(* IEC 61131-3 sources: tuk_project/src/control_systems/implementation/Old, 7 files *)

(* ---- sorting_buffer_assembly.st ---- *)
(****************************************************************************************************************************)
(* SORTING FUNCTION BLOCK *)
(****************************************************************************************************************************)

FUNCTION_BLOCK sorting
  (*==========================================================================================*)
  (* INPUTS AND OUTPUTS *)
  (*==========================================================================================*)

  (* INPUT *)
  (*------------------------------------------------------------*)
  VAR_INPUT
    S_AL1 : BOOL;
    S_BIN_1 : BOOL;
    S_AL1_BL : BOOL;
    CS_AL1_W : INT;
    RUNNING : BOOL;
  END_VAR

  (* OUTPUT *)
  (*------------------------------------------------------------*)
  VAR_OUTPUT
    SB_AL1 : BOOL;
    PUWS_AL1_1_PLUS : BOOL;
    PUWS_AL1_1_RT : BOOL;
    CS_AL1_PLUS : BOOL;
  END_VAR

  (* PLACES *)
  (*------------------------------------------------------------*)
  VAR_EXTERNAL
    P0 : BOOL;
    P1 : BOOL;
    P2 : BOOL;
    P3 : BOOL;
    P4 : BOOL;
    PB : BOOL;
    P5 : BOOL;
    P6 : BOOL;
    BIN1 : BOOL;
    BIN2 : BOOL;
    P_LID : BOOL;
    P_BASE : BOOL;
    STABLE : BOOL;
  END_VAR

  (* OTHERS *)
  (*------------------------------------------------------------*)
  VAR
    timer_1_P2 : TON;
    timer_1_P3 : TON;
  END_VAR

  timer_1_P2(IN:= P2, PT:= T#1000ms);
  timer_1_P3(IN:= P3, PT:= T#1000ms);

  STABLE:= 0;

  IF NOT RUNNING THEN
    P0:= 1;
    P1:= 1;
    P2:= 0;
    P3:= 0;
    P4:= 0;
    PB:= 0;
    BIN1:= 1;
    BIN2:= 0;
    P5:= 0;
    P6:= 0;
    P_LID:= 0;
    P_BASE:= 0;
  END_IF;

  P0:= 1;

  (*==========================================================================================*)
  (* TRANSITIONS *)
  (*==========================================================================================*)
  WHILE STABLE= 0 DO
    STABLE:= 1;
    (*T0112*)
    IF P0 AND P1 AND S_AL1 AND NOT P2 THEN
      P0:= 0;
      P1:= 0;
      P2:= 1;
      STABLE:= 0;
    END_IF;

    (*T23*)
    IF P2 AND timer_1_P2.Q AND NOT P3 THEN
      P2:= 0;
      P3:= 1;
      STABLE:= 0;
    END_IF;

    (*T34*)
    IF P3 AND timer_1_P3.Q AND NOT P4 THEN
      P3:= 0;
      P4:= 1;
    END_IF;

    (*T4B*)
    IF P4 AND ( (CS_AL1_W < 200) OR (CS_AL1_W > 400) ) AND NOT PB THEN
      P4:= 0;
      PB:= 1;
      STABLE:= 0;
    END_IF;

    (*T4B2*)
    IF PB AND BIN1 AND S_BIN_1 AND NOT BIN2 AND NOT P1 THEN
      PB:= 0;
      BIN1:= 0;
      BIN2:= 1;
      P1:= 1;
      STABLE:= 0;
    END_IF;

    (*TB21*)
    IF BIN2 AND NOT S_BIN_1 AND NOT BIN1 THEN
      BIN2:= 0;
      BIN1:= 1;
      STABLE:= 0;
    END_IF;

    (*T45*)
    IF P4 AND ( (CS_AL1_W > 200) AND (CS_AL1_W <= 300) ) AND NOT P5 THEN
      P4:= 0;
      P5:= 1;
      STABLE:= 0;
    END_IF;

    (*T46*)
    IF P4 AND ( (CS_AL1_W > 300) AND (CS_AL1_W <= 400) ) AND NOT P6 THEN
      P4:= 0;
      P6:= 1;
      STABLE:= 0;
    END_IF;

    (*T57*)
    IF P5 AND S_AL1_BL AND NOT P_LID AND NOT P1 THEN
      P5:= 0;
      P_LID:= 1;
      P1:= 1;
      STABLE:= 0;
    END_IF;

    (*T67*)
    IF P6 AND S_AL1_BL AND NOT P_BASE AND NOT P1 THEN
      P6:= 0;
      P_BASE:= 1;
      P1:= 1;
      STABLE:= 0;
    END_IF;

  END_WHILE;

  (*==========================================================================================*)
  (* OUTPUTS *)
  (*==========================================================================================*)
  (*SET SB_AL1*)
  IF P3 OR P4 OR PB OR P5 OR P6 THEN
    SB_AL1:= 1;
  END_IF;
  (*RESET SB_AL1*)
  IF P1 OR P2 THEN
    SB_AL1:= 0;
  END_IF;

  (*SET PUWS_AL1_1_PLUS*)
  IF PB OR P5 OR P6 THEN
    PUWS_AL1_1_PLUS:= 1;
  END_IF;

  (*RESET PUWS_AL1_1_PLUS*)
  IF P1 OR P2 OR P3 OR P4 THEN
    PUWS_AL1_1_PLUS:= 0;
  END_IF;

  (*SET PUWS_AL1_1_RT*)
  IF P5 OR P6 THEN
    PUWS_AL1_1_RT:= 1;
  END_IF;

  (*RESET PUWS_AL1_1_RT*)
  IF P1 OR P2 OR P3 OR P4 OR PB THEN
    PUWS_AL1_1_RT:= 0;
  END_IF;

  (*SET CS_AL1_PLUS*)
  IF P1 OR P2 OR P5 OR P6 OR PB THEN
    CS_AL1_PLUS:= 1;
  END_IF;

  (*RESET CS_AL1_PLUS*)
  IF P3 OR P4 THEN
    CS_AL1_PLUS:= 0;
  END_IF;

END_FUNCTION_BLOCK

(****************************************************************************************************************************)
(* BASE BUFFER FUNCTION BLOCK *)
(****************************************************************************************************************************)

FUNCTION_BLOCK base_buffer
  (*==========================================================================================*)
  (* INPUTS AND OUTPUTS *)
  (*==========================================================================================*)

  (* INPUT *)
  (*------------------------------------------------------------*)
  VAR_INPUT
    S_AL1_B : BOOL;
    P_AL1_B_FT : BOOL;
    P_AL1_B_BK : BOOL;
    S_AL1_B1 : BOOL;
    S_AL1_B2 : BOOL;
    S_AL1_B3 : BOOL;
    S_AL1_LP : BOOL;
    RUNNING : BOOL;
  END_VAR

  (* OUTPUT *)
  (*------------------------------------------------------------*)
  VAR_OUTPUT
    P_AL1_B : BOOL;
    SB_AL1_B1 : BOOL;
    SB_AL1_B2 : BOOL;
    SB_AL1_B3 : BOOL;
    STABLE : BOOL;
  END_VAR

  (* PLACES *)
  (*------------------------------------------------------------*)
  VAR_EXTERNAL
    P_BASE : BOOL;
    PB1 : BOOL;
    PUSH_B : BOOL;
    PB2 : BOOL;
    PB23 : BOOL;
    PB3 : BOOL;
    PB4 : BOOL;
    PB5 : BOOL;
    PB6 : BOOL;
    PB7 : BOOL;
    PB8 : BOOL;
    PBF1 : BOOL;
    PBF2 : BOOL;
    PBF3 : BOOL;
    PBF4 : BOOL;
  END_VAR

  (* OTHERS *)
  (*------------------------------------------------------------*)
  VAR
    timer_1_TB1 : TON;
  END_VAR

  timer_1_TB1(IN:= PB1, PT:= T#900ms);

  STABLE:= 0;

  IF NOT RUNNING THEN
    P_BASE:= 0;
    PB1:= 0;
    PUSH_B:= 1;
    PB2:= 0;
    PB23:= 0;
    PB3:= 0;
    PB4:= 0;
    PB5:= 0;
    PB6:= 0;
    PB7:= 0;
    PB8:= 0;
    PBF1:=1;
    PBF2:=1;
    PBF3:=1;
    PBF4:=1;

  END_IF;

  (*==========================================================================================*)
  (* TRANSITIONS *)
  (*==========================================================================================*)
  WHILE STABLE= 0 DO
    STABLE:= 1;

    (*TB0*)
    IF P_BASE AND S_AL1_B AND NOT PB1 THEN
      P_BASE:=0;
      PB1:=1;
      STABLE:=0;
    END_IF;

    (*TB1*)
    IF PB1 AND PUSH_B AND timer_1_TB1.Q AND NOT PB2 THEN
      PB1:=0;
      PUSH_B:=0;
      PB2:=1;
      STABLE:=0;
    END_IF;

    (*TB23*)
    IF PB2 AND P_AL1_B_FT AND NOT PB23 THEN
      PB2:=0;
      PB23:=1;
      STABLE:=0;
    END_IF;

    (*TB2*)
    IF PB23 AND P_AL1_B_FT AND NOT PB3 THEN
      PB23:=0;
      PB3:=1;
      STABLE:=0;
    END_IF;

    (*TB3*)
    IF PB3 AND P_AL1_B_BK AND NOT PB4 AND NOT PUSH_B THEN
      PB3:=0;
      PB4:=1;
      PUSH_B:=1;
      STABLE:=0;
    END_IF;

    (*TB4*)
    IF PB4 AND PBF1 AND S_AL1_B1 AND NOT PB5 THEN
      PB4:=0;
      PBF1:=0;
      PB5:=1;
      STABLE:=0;
    END_IF;

    (*TB5*)
    IF PB5 AND PBF2 AND S_AL1_B2 AND NOT PB6 AND NOT PBF1 THEN
      PB5:=0;
      PBF2:=0;
      PB6:=1;
      PBF1:=1;
      STABLE:=0;
    END_IF;

    (*TB6*)
    IF PB6 AND PBF3 AND S_AL1_B3 AND  NOT PB7 AND NOT PBF2 THEN
      PB6:=0;
      PBF3:=0;
      PB7:=1;
      PBF2:=1;
      STABLE:=0;
    END_IF;

    (*TB7*)
    IF PB7 AND PBF4 AND S_AL1_LP AND NOT PB8 THEN
      PB7:=0;
      PBF4:=0;
      PB8:=1;
      STABLE:=0;
    END_IF;

  END_WHILE;

  (*==========================================================================================*)
  (* OUTPUTS *)
  (*==========================================================================================*)
  (*P_AL1_B*)
  IF PB2 OR PB23 THEN
    P_AL1_B:=1;
  END_IF;
  IF P_BASE OR PB1 OR PB3 THEN
    P_AL1_B:=0;
  END_IF;

  (*SB_AL1_B1*)
  IF PB5 THEN
    SB_AL1_B1:=1;
  END_IF;
  IF PBF1 THEN
    SB_AL1_B1:=0;
  END_IF;

  (*SB_AL1_B2*)
  IF PB6 THEN
    SB_AL1_B2:=1;
  END_IF;
  IF PBF2 THEN
    SB_AL1_B2:=0;
  END_IF;

  (*SB_AL1_B3*)
  IF PB7 THEN
    SB_AL1_B3:=1;
  END_IF;
  IF PBF3 THEN
    SB_AL1_B3:=0;
  END_IF;

END_FUNCTION_BLOCK

(****************************************************************************************************************************)
(* LID BUFFER FUNCTION BLOCK *)
(****************************************************************************************************************************)

FUNCTION_BLOCK lid_buffer
  (*==========================================================================================*)
  (* INPUTS AND OUTPUTS *)
  (*==========================================================================================*)

  (* INPUT *)
  (*------------------------------------------------------------*)
  VAR_INPUT
    S_AL1_L : BOOL;
    P_AL1_L_FT : BOOL;
    P_AL1_L_BK : BOOL;
    S_AL1_L1 : BOOL;
    S_AL1_L2 : BOOL;
    S_AL1_L3 : BOOL;
    S_AL1_RP : BOOL;
    RUNNING : BOOL;
  END_VAR

  (* OUTPUT *)
  (*------------------------------------------------------------*)
  VAR_OUTPUT
    P_AL1_L : BOOL;
    SB_AL1_L1 : BOOL;
    SB_AL1_L2 : BOOL;
    SB_AL1_L3 : BOOL;
    STABLE : BOOL;
  END_VAR

  (* PLACES *)
  (*------------------------------------------------------------*)
  VAR_EXTERNAL
    P_LID : BOOL;
    PL1 : BOOL;
    PUSH_L : BOOL;
    PL2 : BOOL;
    PL23 : BOOL;
    PL3 : BOOL;
    PL4 : BOOL;
    PL5 : BOOL;
    PL6 : BOOL;
    PL7 : BOOL;
    PL8 : BOOL;
    PLF1 : BOOL;
    PLF2 : BOOL;
    PLF3 : BOOL;
    PLF4 : BOOL;
  END_VAR

  (* OTHERS *)
  (*------------------------------------------------------------*)
  VAR
    timer_1_TL1 : TON;
  END_VAR

  timer_1_TL1(IN:= PL1, PT:= T#900ms);

  STABLE:= 0;

  IF NOT RUNNING THEN
    P_LID:= 0;
    PL1:= 0;
    PUSH_L:= 1;
    PL2:= 0;
    PL23:= 0;
    PL3:= 0;
    PL4:= 0;
    PL5:= 0;
    PL6:= 0;
    PL7:= 0;
    PL8:= 0;
    PLF1:=1;
    PLF2:=1;
    PLF3:=1;
    PLF4:=1;

  END_IF;

  (*==========================================================================================*)
  (* TRANSITIONS *)
  (*==========================================================================================*)
  WHILE STABLE= 0 DO
    STABLE:= 1;

    (*TL0*)
    IF P_LID AND S_AL1_L AND NOT PL1 THEN
      P_LID:=0;
      PL1:=1;
      STABLE:=0;
    END_IF;

    (*TL1*)
    IF PL1 AND PUSH_L AND timer_1_TL1.Q AND NOT PL2 THEN
      PL1:=0;
      PUSH_L:=0;
      PL2:=1;
      STABLE:=0;
    END_IF;

    (*TL23*)
    IF PL2 AND P_AL1_L_FT AND NOT PL23 THEN
      PL2:=0;
      PL23:=1;
      STABLE:=0;
    END_IF;

    (*TL2*)
    IF PL23 AND P_AL1_L_FT AND NOT PL3 THEN
      PL23:=0;
      PL3:=1;
      STABLE:=0;
    END_IF;

    (*TL3*)
    IF PL3 AND P_AL1_L_BK AND NOT PL4 AND NOT PUSH_L THEN
      PL3:=0;
      PL4:=1;
      PUSH_L:=1;
      STABLE:=0;
    END_IF;

    (*TL4*)
    IF PL4 AND PLF1 AND S_AL1_L1 AND NOT PL5 THEN
      PL4:=0;
      PLF1:=0;
      PL5:=1;
      STABLE:=0;
    END_IF;

    (*TL5*)
    IF PL5 AND PLF2 AND S_AL1_L2 AND NOT PL6 AND NOT PLF1 THEN
      PL5:=0;
      PLF2:=0;
      PL6:=1;
      PLF1:=1;
      STABLE:=0;
    END_IF;

    (*TL6*)
    IF PL6 AND PLF3 AND S_AL1_L3 AND  NOT PL7 AND NOT PLF2 THEN
      PL6:=0;
      PLF3:=0;
      PL7:=1;
      PLF2:=1;
      STABLE:=0;
    END_IF;

    (*TL7*)
    IF PL7 AND PLF4 AND S_AL1_RP AND NOT PL8 THEN
      PL7:=0;
      PLF4:=0;
      PL8:=1;
      STABLE:=0;
    END_IF;

  END_WHILE;

  (*==========================================================================================*)
  (* OUTPUTS *)
  (*==========================================================================================*)
  (*P_AL1_L*)
  IF PL2 OR PL23 THEN
    P_AL1_L:=1;
  END_IF;
  IF P_LID OR PL1 OR PL3 THEN
    P_AL1_L:=0;
  END_IF;

  (*SB_AL1_L1*)
  IF PL5 THEN
    SB_AL1_L1:=1;
  END_IF;
  IF PLF1 THEN
    SB_AL1_L1:=0;
  END_IF;

  (*SB_AL1_L2*)
  IF PL6 THEN
    SB_AL1_L2:=1;
  END_IF;
  IF PLF2 THEN
    SB_AL1_L2:=0;
  END_IF;

  (*SB_AL1_L3*)
  IF PL7 THEN
    SB_AL1_L3:=1;
  END_IF;
  IF PLF3 THEN
    SB_AL1_L3:=0;
  END_IF;

END_FUNCTION_BLOCK

(****************************************************************************************************************************)
(* ASSEMBLY FUNCTION BLOCK *)
(****************************************************************************************************************************)
FUNCTION_BLOCK assembly
  (*==========================================================================================*)
  (* INPUTS AND OUTPUTS *)
  (*==========================================================================================*)

  (* INPUT *)
  (*------------------------------------------------------------*)
  VAR_INPUT
    AL1_DETECTED : BOOL;
    AL1_X_POS : WORD;
    AL1_Y_POS : WORD;
    AL1_Z_POS : WORD;
    LP_AL1_CLAMPED : BOOL;
    LP_AL1_LIMIT : BOOL;
    RP_AL1_CLAMPED : BOOL;
    RUNNING : BOOL;
  END_VAR

  (* OUTPUT *)
  (*------------------------------------------------------------*)
  VAR_OUTPUT
    AL1_X_SET : WORD;
    AL1_Y_SET : WORD;
    AL1_Z_SET : WORD;
    AL1_GRAB : BOOL;
    RP_AL1_CLAMP : BOOL;
    LP_AL1_RAISE : BOOL;
    LP_AL1_CLAMP : BOOL;
    SB_AL1_B3 : BOOL;
    SB_AL1_L3 : BOOL;
    STABLE : BOOL;
  END_VAR

  (* PLACES *)
  (*------------------------------------------------------------*)
  VAR_EXTERNAL
    PA0 : BOOL;
    PA1 : BOOL;
    PA2 : BOOL;
    PA3 : BOOL;
    PA4 : BOOL;
    PA5 : BOOL;
    PA6 : BOOL;
    PA7 : BOOL;
    PA8 : BOOL;
    PA9 : BOOL;
    PA10 : BOOL;
    PA11 : BOOL;
    PA12 : BOOL;
    PA13 : BOOL;
    PB8 : BOOL;
    PB9 : BOOL;
    PL8 : BOOL;
    PL9 : BOOL;
    PBF3 : BOOL;
    PBF4 : BOOL;
    PLF3 : BOOL;
    PLF4 : BOOL;
  END_VAR

  (* OTHERS *)
  (*------------------------------------------------------------*)
  VAR
    timer_1 : TON;
  END_VAR

  timer_1(IN:= PL9, PT:= T#300ms);

  STABLE:= 0;

  IF NOT RUNNING THEN

    PB9:=0;
    PL9:=0;
    PA0:=1;
    PA1:=0;
    PA2:=0;
    PA3:=0;
    PA4:=0;
    PA5:=0;
    PA6:=0;
    PA7:=0;
    PA8:=0;
    PA9:=0;
    PA10:=0;
    PA11:=0;
    PA12:=0;
    PA13:=0;
  END_IF;

  (*==========================================================================================*)
  (* TRANSITIONS *)
  (*==========================================================================================*)
  WHILE STABLE=0 DO

    STABLE:=1;

    (*TB8*)
    IF PB8 AND LP_AL1_CLAMPED AND NOT PB9 THEN
      PB8:=0;
      PB9:=1;
      STABLE:=0;
    END_IF;

    (*TL8*)
    IF PL8 AND RP_AL1_CLAMPED AND NOT PL9 THEN
      PL8:=0;
      PL9:=1;
      STABLE:=0;
    END_IF;

    (*TA0*)
    IF PL9 AND timer_1.Q AND PA0 AND RP_AL1_CLAMPED AND NOT AL1_DETECTED AND NOT PA1 THEN
      PL9:=0;
      PA0:=0;
      PA1:=1;
      STABLE:=0;
    END_IF;

    (*TA1*)
    IF PA1 AND AL1_X_POS>798 AND AL1_X_POS<802 AND AL1_Y_POS>148 AND AL1_Y_POS<152 AND NOT PA2 THEN
      PA1:=0;
      PA2:=1;
      STABLE:=0;
    END_IF;

    (*TA2*)
    IF PA2 AND AL1_Z_POS>798 AND AL1_Z_POS<802 AND NOT PA3 THEN
      PA2:=0;
      PA3:=1;
      STABLE:=0;
    END_IF;

    (*TA3*)
    IF PA3 AND NOT RP_AL1_CLAMPED AND NOT PA4 THEN
      PA3:=0;
      PA4:=1;
      STABLE:=0;
    END_IF;

    (*TA4*)
    IF PA4 AND AL1_Z_POS>398 AND AL1_Z_POS<402 AND NOT PA5 AND NOT PLF3 AND NOT PLF4 THEN
      PA4:=0;
      PA5:=1;
      PLF3:=1;
      PLF4:=1;
      STABLE:=0;
    END_IF;

    (*TA5*)
    IF PA5 AND PB9 AND AL1_DETECTED AND LP_AL1_CLAMPED AND AL1_X_POS>208 AND AL1_X_POS<212 AND AL1_Y_POS>148 AND AL1_Y_POS<152 AND NOT PA6 THEN
      PA5:=0;
      PB9:=0;
      PA6:=1;
      STABLE:=0;
    END_IF;

    (*TA6*)
    IF PA6 AND AL1_Z_POS>810 AND AL1_Z_POS<820 AND NOT PA7 THEN
      PA6:=0;
      PA7:=1;
      STABLE:=0;
    END_IF;

    (*TA7*)
    IF PA7 AND AL1_Z_POS>398 AND AL1_Z_POS<402 AND NOT PA8 THEN
      PA7:=0;
      PA8:=1;
      STABLE:=0;
    END_IF;

    (*TA8*)
    IF PA8 AND NOT LP_AL1_CLAMPED AND NOT PA9 THEN
      PA8:=0;
      PA9:=1;
      STABLE:=0;
    END_IF;

    (*TA9*)
    IF PA9 AND NOT LP_AL1_LIMIT AND NOT PA10 THEN
      PA9:=0;
      PA10:=1;
      STABLE:=0;
    END_IF;

    (*TA10*)
    IF PA10 AND LP_AL1_LIMIT AND NOT PA11 THEN
      PA10:=0;
      PA11:=1;
      STABLE:=0;
    END_IF;

    (*TA11*)
    IF PA11 AND NOT LP_AL1_LIMIT AND NOT PA12 THEN
      PA11:=0;
      PA12:=1;
      STABLE:=0;
    END_IF;

    (*TA12*)
    IF PA12 AND LP_AL1_LIMIT AND NOT PA13 AND NOT PA0 AND NOT PBF3 AND NOT PBF4 THEN
      PA12:=0;
      PA13:=1;
      PA0:=1;
      PBF3:=1;
      PBF4:=1;
      STABLE:=0;
    END_IF;

  END_WHILE;

  (*==========================================================================================*)
  (* OUTPUTS *)
  (*==========================================================================================*)

  (*LP_AL1_CLAMP*)
  IF PB8 OR PB9 THEN
    LP_AL1_CLAMP:=1;
  END_IF;
  IF PBF4 THEN
    LP_AL1_CLAMP:=0;
  END_IF;

  (*RP_AL1_CLAMP*)
  IF PL8 OR PL9 THEN
    RP_AL1_CLAMP:=1;
  END_IF;
  IF PLF4 THEN
    RP_AL1_CLAMP:=0;
  END_IF;

  (*MOVE GRABBER TO LID POSITION*)
  IF PA1 THEN
    AL1_X_SET:=800;
    AL1_Y_SET:=150;
  END_IF;

  (*GRABBER DOWN TO PICK LID*)
  IF PA2 THEN
    AL1_Z_SET:= 800;
  END_IF;

  (*GRAB LID*)
  IF PA3 OR PA4 OR PA5 OR PA6 THEN
    AL1_GRAB:=1;
  END_IF;

  (*RAISE GRABBER A LITTLE*)
  IF PA0 OR PA4 OR PA7 THEN
    AL1_Z_SET:=400;
  END_IF;

  (*MOVE GRABBER TO BASE POSITION*)
  IF PA0 OR PA5 THEN
    AL1_X_SET:=210;
    AL1_Y_SET:=150;
  END_IF;

  (*LOWER LID TO FIT ON BASE*)
  IF PA6 THEN
    AL1_Z_SET:=818;
  END_IF;

  (*RELEASE LID*)
  IF PA0 OR PA1 OR PA2 OR PA7 OR PA8 OR PA9 OR PA10 OR PA11 OR PA12 THEN
    AL1_GRAB:=0;
  END_IF;

  (*LID CLAMP*)
  IF PA1 OR PA2 THEN
    RP_AL1_CLAMP:=1;
  END_IF;

  IF PA3 OR PA4 OR PLF4 THEN
    RP_AL1_CLAMP:=0;
  END_IF;

  (*BASE CLAMP*)
  IF PA8 OR PA9 OR PA10 OR PA11 OR PA12 THEN
    LP_AL1_CLAMP:=0;
  END_IF;

  IF PB9 OR PA6 OR PA7 THEN
    LP_AL1_CLAMP:=1;
  END_IF;

  (*RAISE BASE CLAMP*)
  IF PA0 OR PA1 OR PA2 OR PA3 OR PA4 OR PA5 OR PA6 OR PA7 OR PA8 OR PA11 OR PA12 THEN
    LP_AL1_RAISE:=0;
  END_IF;

  IF PA9 OR PA10 THEN
    LP_AL1_RAISE:=1;
  END_IF;

  (* OUTPUTS OF PLACES FROM OTHER STAGES *)
  (*LP_AL1_CLAMP*)
  (*IF PB9 THEN
    LP_AL1_CLAMP:=1;
  END_IF;
  IF PBF4 THEN
    LP_AL1_CLAMP:=0;
  END_IF;

  (*SB_AL1_B3
  IF PBF3 THEN
    SB_AL1_B3:=0;
  END_IF;

  (*SB_AL1_L3
  IF PLF3 THEN
    SB_AL1_L3:=0;
  END_IF;

  (*RP_AL1_CLAMP
  IF PL9 THEN
    RP_AL1_CLAMP:=1;
  END_IF;
  IF PLF4 THEN
    RP_AL1_CLAMP:=0;
  END_IF;  *)

END_FUNCTION_BLOCK

(****************************************************************************************************************************)
(* MAIN PROGRAM *)
(****************************************************************************************************************************)

PROGRAM sorting_buffer_assembly

  (****************************************************************************************************************************)
  (* VARIABLE DECLARATION *)
  (****************************************************************************************************************************)

  (*==========================================================================================*)
  (* INPUTS AND OUTPUTS *)
  (*==========================================================================================*)

  (* SORTING *)
  (*------------------------------------------------------------*)
  VAR
    (* INPUTS *)
    S_AL1 AT %IX102.0 : BOOL;
    S_BIN_1 AT %IX102.1 : BOOL;
    S_AL1_BL AT %IX102.2 : BOOL;
    CS_AL1_W AT %IW100 : INT;

    (* OUTPUTS *)
    SB_AL1 AT %QX101.2 : BOOL;
    PUWS_AL1_1_PLUS AT %QX101.3 : BOOL;
    PUWS_AL1_1_RT AT %QX101.4 : BOOL;
    CS_AL1_PLUS AT %QX101.5 : BOOL;
  END_VAR

  (* BUFFER *)
  (*------------------------------------------------------------*)
  VAR
    (* INPUTS *)
    S_AL1_B AT %IX100.0 : BOOL;
    P_AL1_B_FT AT %IX100.1 : BOOL;
    P_AL1_B_BK AT %IX100.2 : BOOL;
    S_AL1_B1 AT %IX100.3 : BOOL;
    S_AL1_B2 AT %IX100.4 : BOOL;
    S_AL1_B3 AT %IX100.5 : BOOL;
    LP_AL1_CLAMPED AT %IX100.6 : BOOL;
    S_AL1_LP AT %IX100.7 : BOOL;
    S_AL1_L AT %IX101.0 : BOOL;
    P_AL1_L_FT AT %IX101.1 : BOOL;
    P_AL1_L_BK AT %IX101.2 : BOOL;
    S_AL1_L1 AT %IX101.3 : BOOL;
    S_AL1_L2 AT %IX101.4 : BOOL;
    S_AL1_L3 AT %IX101.5 : BOOL;
    RP_AL1_CLAMPED AT %IX101.6 : BOOL;
    S_AL1_RP AT %IX101.7 : BOOL;

    (* OUTPUTS *)
    P_AL1_B AT %QX100.0 : BOOL;
    SB_AL1_B1 AT %QX100.1 : BOOL;
    SB_AL1_B2 AT %QX100.2 : BOOL;
    SB_AL1_B3 AT %QX100.3 : BOOL;
    LP_AL1_CLAMP AT %QX100.4 : BOOL;
    P_AL1_L AT %QX100.5 : BOOL;
    SB_AL1_L1 AT %QX100.6 : BOOL;
    SB_AL1_L2 AT %QX100.7 : BOOL;
    SB_AL1_L3 AT %QX101.0 : BOOL;
    RP_AL1_CLAMP AT %QX101.1 : BOOL;

  END_VAR

  (* ASSEMBLY *)
  (*------------------------------------------------------------*)
  VAR
    (* INPUTS *)
    AL1_DETECTED AT %IX102.3 : BOOL;
    LP_AL1_LIMIT AT %IX102.4 : BOOL;
    AL1_X_POS AT %IW101 : WORD;
    AL1_Y_POS AT %IW102 : WORD;
    AL1_Z_POS AT %IW103 : WORD;

    (* OUTPUTS *)
    AL1_GRAB AT %QX101.6 : BOOL;
    LP_AL1_RAISE AT %QX101.7 : BOOL;
    AL1_X_SET AT %QW100 : WORD;
    AL1_Y_SET AT %QW101 : WORD;
    AL1_Z_SET AT %QW102 : WORD;

  END_VAR

  (* OTHERS *)
  (*------------------------------------------------------------*)
  VAR
    (* RUNNING *)
    RUNNING AT %IX102.7 : BOOL;
  END_VAR

  (*==========================================================================================*)
  (* PLACES *)
  (*==========================================================================================*)
  (* ASSEMBLY *)
  (*------------------------------------------------------------*)
  VAR_EXTERNAL

    PA0 : BOOL;
    PA1 : BOOL;
    PA2 : BOOL;
    PA3 : BOOL;
    PA4 : BOOL;
    PA5 : BOOL;
    PA6 : BOOL;
    PA7 : BOOL;
    PA8 : BOOL;
    PA9 : BOOL;
    PA10 : BOOL;
    PA11 : BOOL;
    PA12 : BOOL;
    PA13 : BOOL;
    PL9 : BOOL;
    PB9 : BOOL;
    PBF3 : BOOL;
    PBF4 : BOOL;
    PLF3 : BOOL;
    PLF4 : BOOL;
  END_VAR
  (*==========================================================================================*)
  (* OTHERS *)
  (*==========================================================================================*)
  VAR_EXTERNAL
    STABLE : BOOL;
  END_VAR

  (****************************************************************************************************************************)
  (* VARIABLE INITIALIZATION *)
  (****************************************************************************************************************************)

  (*==========================================================================================*)
  (* FUNTION BLOCKS *)
  (*==========================================================================================*)
  VAR
    sorting0 : sorting;
    base_buffer0 : base_buffer;
    lid_buffer0 : lid_buffer;
    assembly0 : assembly;
  END_VAR

  (*==========================================================================================*)
  (* PLACES *)
  (*==========================================================================================*)

  (****************************************************************************************************************************)
  (* FUNCTION BLOCKS *)
  (****************************************************************************************************************************)

  (* SORTING *)
  (*------------------------------------------------------------*)
  sorting0(
    S_AL1:=S_AL1, S_BIN_1:=S_BIN_1, S_AL1_BL:=S_AL1_BL,
    CS_AL1_W:=CS_AL1_W, RUNNING:=RUNNING,

    SB_AL1=>SB_AL1, PUWS_AL1_1_PLUS=>PUWS_AL1_1_PLUS,
    PUWS_AL1_1_RT=>PUWS_AL1_1_RT, CS_AL1_PLUS=>CS_AL1_PLUS
  );

  (* BASE BUFFER *)
  (*------------------------------------------------------------*)
  base_buffer0(
    S_AL1_B:=S_AL1_B, P_AL1_B_FT:=P_AL1_B_FT, P_AL1_B_BK:=P_AL1_B_BK,
    S_AL1_B1:=S_AL1_B1, S_AL1_B2:=S_AL1_B2, S_AL1_B3:=S_AL1_B3,
    S_AL1_LP:=S_AL1_LP, (*LP_AL1_CLAMPED:=LP_AL1_CLAMPED,*) RUNNING:=RUNNING,

    P_AL1_B=>P_AL1_B, SB_AL1_B1=>SB_AL1_B1, SB_AL1_B2=>SB_AL1_B2,
    SB_AL1_B3=>SB_AL1_B3, STABLE=>STABLE (*, LP_AL1_CLAMP=>LP_AL1_CLAMP*)
  );

  (* LID BUFFER *)
  (*------------------------------------------------------------*)
  lid_buffer0(
    S_AL1_L:=S_AL1_L, P_AL1_L_FT:=P_AL1_L_FT, P_AL1_L_BK:=P_AL1_L_BK,
    S_AL1_L1:=S_AL1_L1, S_AL1_L2:=S_AL1_L2, S_AL1_L3:=S_AL1_L3,
    S_AL1_RP:=S_AL1_RP, (*RP_AL1_CLAMPED:=RP_AL1_CLAMPED,*) RUNNING:=RUNNING,

    P_AL1_L=>P_AL1_L, SB_AL1_L1=>SB_AL1_L1, SB_AL1_L2=>SB_AL1_L2,
    SB_AL1_L3=>SB_AL1_L3, STABLE=>STABLE (*, RP_AL1_CLAMP=>RP_AL1_CLAMP*)
  );

  (* ASSEMBLY *)
  (*------------------------------------------------------------*)
  assembly0(
    RP_AL1_CLAMPED:=RP_AL1_CLAMPED, AL1_DETECTED:=AL1_DETECTED,
    AL1_X_POS:=AL1_X_POS, AL1_Y_POS:=AL1_Y_POS, AL1_Z_POS:=AL1_Z_POS,
    LP_AL1_CLAMPED:=LP_AL1_CLAMPED, LP_AL1_LIMIT:=LP_AL1_LIMIT,
    RUNNING:=RUNNING,

    AL1_X_SET=>AL1_X_SET, AL1_Y_SET=>AL1_Y_SET, AL1_Z_SET=>AL1_Z_SET,
    AL1_GRAB=>AL1_GRAB, RP_AL1_CLAMP=>RP_AL1_CLAMP, LP_AL1_CLAMP=>LP_AL1_CLAMP,
    LP_AL1_RAISE=>LP_AL1_RAISE, STABLE=>STABLE (*,SB_AL1_B3=>SB_AL1_B3, SB_AL1_L3=>SB_AL1_L3*)
  );

END_PROGRAM

CONFIGURATION Config0

  (*==========================================================================================*)
  (* PLACES *)
  (*==========================================================================================*)

  (* SORTING *)
  (*------------------------------------------------------------*)
  VAR_GLOBAL
    P0 AT %QX103.0 : BOOL;
    P1 AT %QX103.1 : BOOL;
    P2 AT %QX103.2 : BOOL;
    P3 AT %QX103.3 : BOOL;
    P4 AT %QX103.4 : BOOL;
    PB AT %QX103.5 : BOOL;
    P5 AT %QX103.6 : BOOL;
    P6 AT %QX103.7 : BOOL;
    BIN1 AT %QX104.0 : BOOL;
    BIN2 AT %QX104.1 : BOOL;
    P_LID AT %QX104.2 : BOOL;
    P_BASE AT %QX104.3 : BOOL;
  END_VAR

  (* BUFFER *)
  (*------------------------------------------------------------*)
  VAR_GLOBAL
    PB1 AT %QX105.1 : BOOL;
    PUSH_B AT %QX105.2 : BOOL;
    PB2 AT %QX105.3 : BOOL;
    PB23 AT %QX105.4 : BOOL;
    PB3 AT %QX105.5 : BOOL;
    PB4 AT %QX105.6 : BOOL;
    PB5 AT %QX105.7 : BOOL;
    PB6 AT %QX106.0 : BOOL;
    PB7 AT %QX106.1 : BOOL;
    PB8 AT %QX106.2 : BOOL;
    PB9 AT %QX106.3 : BOOL;
    PBF1 AT %QX106.4 : BOOL;
    PBF2 AT %QX106.5 : BOOL;
    PBF3 AT %QX106.6 : BOOL;
    PBF4 AT %QX106.7 : BOOL;
    PL1 AT %QX107.1 : BOOL;
    PL2 AT %QX107.2 : BOOL;
    PUSH_L AT %QX107.3 : BOOL;
    PL23 AT %QX107.4 : BOOL;
    PL3 AT %QX107.5 : BOOL;
    PL4 AT %QX107.6 : BOOL;
    PL5 AT %QX107.7 : BOOL;
    PL6 AT %QX108.0 : BOOL;
    PL7 AT %QX108.1 : BOOL;
    PL8 AT %QX108.2 : BOOL;
    PL9 AT %QX108.3 : BOOL;
    PLF1 AT %QX108.4 : BOOL;
    PLF2 AT %QX108.5 : BOOL;
    PLF3 AT %QX108.6 : BOOL;
    PLF4 AT %QX108.7 : BOOL;
  END_VAR

  (* ASSEMBLY *)
  (*------------------------------------------------------------*)
  VAR_GLOBAL
    PA0 AT %QX109.0 : BOOL;
    PA1 AT %QX109.1 : BOOL;
    PA2 AT %QX109.2 : BOOL;
    PA3 AT %QX109.3 : BOOL;
    PA4 AT %QX109.4 : BOOL;
    PA5 AT %QX109.5 : BOOL;
    PA6 AT %QX109.6 : BOOL;
    PA7 AT %QX109.7 : BOOL;
    PA8 AT %QX110.0 : BOOL;
    PA9 AT %QX110.1 : BOOL;
    PA10 AT %QX110.2 : BOOL;
    PA11 AT %QX110.3 : BOOL;
    PA12 AT %QX110.4 : BOOL;
    PA13 AT %QX110.5 : BOOL;
  END_VAR

  (*==========================================================================================*)
  (* OTHERS *)
  (*==========================================================================================*)
  VAR_GLOBAL
    STABLE AT %QX510.0 : BOOL;
  END_VAR

  RESOURCE Res0 ON PLC
    TASK task0(INTERVAL := T#20ms,PRIORITY := 0);
    PROGRAM instance0 WITH task0 : sorting_buffer_assembly;
  END_RESOURCE
END_CONFIGURATION

(* ---- assembly.st ---- *)
PROGRAM assembly
  VAR
    RP_AL1_CLAMPED AT %IX100.0 : BOOL;
    AL1_DETECTED AT %IX100.1 : BOOL;
    LP_AL1_CLAMPED AT %IX100.2 : BOOL;
    LP_AL1_LIMIT AT %IX100.3 : BOOL;
    RUNNING AT %IX100.4 : BOOL;
    AL1_X_POS AT %IW100 : WORD;
    AL1_Y_POS AT %IW101 : WORD;
    AL1_Z_POS AT %IW102 : WORD;
    AL1_GRAB AT %QX100.0 : BOOL;
    RP_AL1_CLAMP AT %QX100.1 : BOOL;
    LP_AL1_CLAMP AT %QX100.2 : BOOL;
    LP_AL1_RAISE AT %QX100.3 : BOOL;
    AL1_X_SET AT %QW100 : WORD;
    AL1_Y_SET AT %QW101 : WORD;
    AL1_Z_SET AT %QW102 : WORD;
    PLF3 AT %QX0.0 : BOOL;
    PLF4 AT %QX0.1 : BOOL;
    PBF3 AT %QX0.2 : BOOL;
    PBF4 AT %QX0.3 : BOOL;
    PL9 AT %QX0.4 : BOOL;
    PB9 AT %QX0.5 : BOOL;
    PA0 AT %QX0.6 : BOOL;
    PA1 AT %QX0.7 : BOOL;
    PA2 AT %QX1.0 : BOOL;
    PA3 AT %QX1.1 : BOOL;
    PA4 AT %QX1.2 : BOOL;
    PA5 AT %QX1.3 : BOOL;
    PA6 AT %QX1.4 : BOOL;
    PA7 AT %QX1.5 : BOOL;
    PA8 AT %QX1.6 : BOOL;
    PA9 AT %QX1.7 : BOOL;
    PA10 AT %QX2.0 : BOOL;
    PA11 AT %QX2.1 : BOOL;
    PA12 AT %QX2.2 : BOOL;
    PA13 AT %QX2.3 : BOOL;
    STABLE AT %QX2.4 : BOOL;
  END_VAR

  IF NOT RUNNING THEN

    PLF3:=0;
    PLF4:=0;
    PBF3:=0;
    PBF4:=0;
    PL9:=1;
    PB9:=1;
    PA0:=1;
    PA1:=0;
    PA2:=0;
    PA3:=0;
    PA4:=0;
    PA5:=0;
    PA6:=0;
    PA7:=0;
    PA8:=0;
    PA9:=0;
    PA10:=0;
    PA11:=0;
    PA12:=0;
    PA13:=0;

  END_IF;

  (*TRANSITIONS*)

  STABLE:=0;

  WHILE STABLE=0 DO

    STABLE:=1;

    (*TA0*)
    IF PL9 AND PA0 AND RP_AL1_CLAMPED AND NOT AL1_DETECTED AND NOT PA1 THEN
      PL9:=0;
      PA0:=0;
      PA1:=1;
      STABLE:=0;
    END_IF;

    (*TA1*)
    IF PA1 AND AL1_X_POS>798 AND AL1_X_POS<802 AND AL1_Y_POS>148 AND AL1_Y_POS<152 AND NOT PA2 THEN
      PA1:=0;
      PA2:=1;
      STABLE:=0;
    END_IF;

    (*TA2*)
    IF PA2 AND AL1_Z_POS>798 AND AL1_Z_POS<802 AND NOT PA3 THEN
      PA2:=0;
      PA3:=1;
      STABLE:=0;
    END_IF;

    (*TA3*)
    IF PA3 AND NOT RP_AL1_CLAMPED AND NOT PA4 THEN
      PA3:=0;
      PA4:=1;
      STABLE:=0;
    END_IF;

    (*TA4*)
    IF PA4 AND AL1_Z_POS>398 AND AL1_Z_POS<402 AND NOT PA5 AND NOT PLF3 AND NOT PLF4 THEN
      PA4:=0;
      PA5:=1;
      PLF3:=1;
      PLF4:=1;
      STABLE:=0;
    END_IF;

    (*TA5*)
    IF PA5 AND PB9 AND AL1_DETECTED AND LP_AL1_CLAMPED AND AL1_X_POS>208 AND AL1_X_POS<212 AND AL1_Y_POS>148 AND AL1_Y_POS<152 AND NOT PA6 THEN
      PA5:=0;
      PB9:=0;
      PA6:=1;
      STABLE:=0;
    END_IF;

    (*TA6*)
    IF PA6 AND AL1_Z_POS>810 AND AL1_Z_POS<820 AND NOT PA7 THEN
      PA6:=0;
      PA7:=1;
      STABLE:=0;
    END_IF;

    (*TA7*)
    IF PA7 AND AL1_Z_POS>398 AND AL1_Z_POS<402 AND NOT PA8 THEN
      PA7:=0;
      PA8:=1;
      STABLE:=0;
    END_IF;

    (*TA8*)
    IF PA8 AND NOT LP_AL1_CLAMPED AND NOT PA9 THEN
      PA8:=0;
      PA9:=1;
      STABLE:=0;
    END_IF;

    (*TA9*)
    IF PA9 AND NOT LP_AL1_LIMIT AND NOT PA10 THEN
      PA9:=0;
      PA10:=1;
      STABLE:=0;
    END_IF;

    (*TA10*)
    IF PA10 AND LP_AL1_LIMIT AND NOT PA11 THEN
      PA10:=0;
      PA11:=1;
      STABLE:=0;
    END_IF;

    (*TA11*)
    IF PA11 AND NOT LP_AL1_LIMIT AND NOT PA12 THEN
      PA11:=0;
      PA12:=1;
      STABLE:=0;
    END_IF;

    (*TA12*)
    IF PA12 AND LP_AL1_LIMIT AND NOT PA13 AND NOT PA0 AND NOT PBF3 AND NOT PBF4 THEN
      PA12:=0;
      PA13:=1;
      PA0:=1;
      PBF3:=1;
      PBF4:=1;
      STABLE:=0;
    END_IF;

  END_WHILE;

  (*OUTPUTS*)
  (*MOVE GRABBER TO LID POSITION*)
  IF PA1 THEN
    AL1_X_SET:=800;
    AL1_Y_SET:=150;
  END_IF;

  (*GRABBER DOWN TO PICK LID*)
  IF PA2 THEN
    AL1_Z_SET:= 800;
  END_IF;

  (*GRAB LID*)
  IF PA3 OR PA4 OR PA5 OR PA6 THEN
    AL1_GRAB:=1;
  END_IF;

  (*RAISE GRABBER A LITTLE*)
  IF PA0 OR PA4 OR PA7 THEN
    AL1_Z_SET:=400;
  END_IF;

  (*MOVE GRABBER TO BASE POSITION*)
  IF PA0 OR PA5 THEN
    AL1_X_SET:=210;
    AL1_Y_SET:=150;
  END_IF;

  (*LOWER LID TO FIT ON BASE*)
  IF PA6 THEN
    AL1_Z_SET:=818;
  END_IF;

  (*RELEASE LID*)
  IF PA0 OR PA1 OR PA2 OR PA7 OR PA8 OR PA9 OR PA10 OR PA11 OR PA12 THEN
    AL1_GRAB:=0;
  END_IF;

  (*LID CLAMP*)
  IF PA1 OR PA2 THEN
    RP_AL1_CLAMP:=1;
  END_IF;

  IF PA3 OR PA4 OR PLF4 THEN
    RP_AL1_CLAMP:=0;
  END_IF;

  (*BASE CLAMP*)
  IF PA8 OR PA9 OR PA10 OR PA11 OR PA12 THEN
    LP_AL1_CLAMP:=0;
  END_IF;

  IF PB9 OR PA6 OR PA7 THEN
    LP_AL1_CLAMP:=1;
  END_IF;

  (*RAISE BASE CLAMP*)
  IF PA0 OR PA1 OR PA2 OR PA3 OR PA4 OR PA5 OR PA6 OR PA7 OR PA8 OR PA11 OR PA12 THEN
    LP_AL1_RAISE:=0;
  END_IF;

  IF PA9 OR PA10 THEN
    LP_AL1_RAISE:=1;
  END_IF;

END_PROGRAM

CONFIGURATION Config0

  RESOURCE Res0 ON PLC
    TASK task0(INTERVAL := T#20ms,PRIORITY := 0);
    PROGRAM instance0 WITH task0 : assembly;
  END_RESOURCE
END_CONFIGURATION

(* ---- demo_factory.st ---- *)
PROGRAM demo_factory
  VAR
    ST_X AT %IX100.0 : BOOL;
    ST_Z AT %IX100.1 : BOOL;
    S_L AT %IX100.2 : BOOL;
    SL_P AT %IX100.3 : BOOL;
    SL_M AT %IX100.4 : BOOL;
    SBC AT %IX100.5 : BOOL;
    SB_P AT %IX100.6 : BOOL;
    SB_M AT %IX100.7 : BOOL;
    RESET AT %IX101.0 : BOOL;
    AT_X AT %QX100.0 : BOOL := 0;
    AT_Z AT %QX100.1 : BOOL := 0;
    AT_G AT %QX100.2 : BOOL := 0;
    AL_C AT %QX100.3 : BOOL := 0;
    AL_M AT %QX100.4 : BOOL := 0;
    RB_M AT %QX100.5 : BOOL := 0;
    AB_C AT %QX100.6 : BOOL := 0;
    AB_M AT %QX100.7 : BOOL := 0;
    (* PLACES ARE SET AS OUTPUTS FOR DEBUGGING *)
    (* PLACES *)                  (* MODBUS ADDERSS *)
    PA1 AT %QX000.0 : BOOL := 1;  (* 0 *)
    PA2 AT %QX000.1 : BOOL := 0;  (* 1 *)
    PA3 AT %QX000.2 : BOOL := 0;  (* 2 *)
    PA4 AT %QX000.3 : BOOL := 0;  (* 3 *)
    PB1 AT %QX000.4 : BOOL := 1;  (* 4 *)
    PB2 AT %QX000.5 : BOOL := 0;  (* 5 *)
    PB3 AT %QX000.6 : BOOL := 0;  (* 6 *)
    PB4 AT %QX000.7 : BOOL := 0;  (* 7 *)
    PC1 AT %QX001.0 : BOOL := 0;  (* 8 *)
    PC2 AT %QX001.1 : BOOL := 0;  (* 9 *)
    PC3 AT %QX001.2 : BOOL := 0;  (* 10 *)
    PC4 AT %QX001.3 : BOOL := 0;  (* 11 *)
    PC5 AT %QX001.4 : BOOL := 0;  (* 12 *)
    PC6 AT %QX001.5 : BOOL := 0;  (* 13 *)
    PC7 AT %QX001.6 : BOOL := 0;  (* 14 *)
    PC8 AT %QX001.7 : BOOL := 0;  (* 15 *)
    PD1 AT %QX002.0 : BOOL := 0;  (* 16 *)
    PD2 AT %QX002.1 : BOOL := 0;  (* 17 *)
    PD3 AT %QX002.2 : BOOL := 0;  (* 18 *)
    PE1 AT %QX002.3 : BOOL := 0;  (* 19 *)
    PE2 AT %QX002.4 : BOOL := 0;  (* 20 *)
    PE3 AT %QX002.5 : BOOL := 0;  (* 21 *)
    PE4 AT %QX002.6 : BOOL := 0;  (* 22 *)
    PE5 AT %QX002.7 : BOOL := 0;  (* 23 *)
    PE6 AT %QX003.0 : BOOL := 0;  (* 24 *)
    PE7 AT %QX003.1 : BOOL := 0;  (* 25 *)
    PF1 AT %QX003.2 : BOOL := 0;  (* 26 *)
    PF2 AT %QX003.3 : BOOL := 0;  (* 27 *)
    PF3 AT %QX003.4 : BOOL := 0;  (* 28 *)
    PF4 AT %QX003.5 : BOOL := 0;  (* 29 *)
    PF5 AT %QX003.6 : BOOL := 1;  (* 30 *)
  END_VAR
  VAR
    TM_1_ta1 : TON;
    TM_1_tc3 : TON;
    TM_1_tb1 : TON;
    TM_1_td3 : TON;
    TM_2_ta3 : TON;
    TM_2_tb3 : TON;
    TM_2_tc5 : TON;
    TM_2_tc6 : TON;
    TM_2_tf1 : TON;
    TM_2_tf2 : TON;
    stable : BOOL := 1;
  END_VAR

  (*============================================================*)
  (* RESET *)
  (*============================================================*)
  IF NOT RESET THEN
      (*OUTPUTS*)
      AT_X:= 0;
      AT_Z:= 0;
      AT_G:= 0;
      AL_C:= 0;
      AL_M:= 0;
      RB_M:= 0;
      AB_C:= 0;
      AB_M:= 0;
      RB_M:= 0;
      (*PLACES*)
      PA1:= 1;
      PA2:= 0;
      PA3:= 0;
      PA4:= 0;
      PB1:= 1;
      PB2:= 0;
      PB3:= 0;
      PB4:= 0;
      PC1:= 0;
      PC2:= 0;
      PC3:= 0;
      PC4:= 0;
      PC5:= 0;
      PC6:= 0;
      PC7:= 0;
      PC8:= 0;
      PD1:= 0;
      PD2:= 0;
      PD3:= 0;
      PE1:= 0;
      PE2:= 0;
      PE3:= 0;
      PE4:= 0;
      PE5:= 0;
      PE6:= 0;
      PE7:= 0;
      PF1:= 0;
      PF2:= 0;
      PF3:= 0;
      PF4:= 0;
      PF5:= 1;
  END_IF;

  (*============================================================*)
  (* TIMERS *)
  (*============================================================*)
  TM_1_ta1(IN:= PA1, PT:= T#2000ms);
  TM_1_tc3(IN:= PC3, PT:= T#2000ms);
  TM_1_tb1(IN:= PB1, PT:= T#2000ms);
  TM_1_td3(IN:= PD3, PT:= T#1000ms);
  TM_2_ta3(IN:= PA3, PT:= T#1000ms);
  TM_2_tb3(IN:= PB3, PT:= T#1000ms);
  TM_2_tc5(IN:= PC5, PT:= T#2000ms);
  TM_2_tc6(IN:= PC6, PT:= T#2000ms);
  TM_2_tf1(IN:= PF1, PT:= T#2000ms);
  TM_2_tf2(IN:= PF2, PT:= T#2000ms);

    stable:= 1;
    (*============================================================*)
    (* TRANSITIONS *)
    (*============================================================*)
    (* Line A *)
    IF PA1 AND NOT PA2 AND TM_1_ta1.Q THEN
      PA1:= 0;
      PA2:= 1;
      stable:= 0;
    END_IF;
    IF PA2 AND NOT PA3 AND SL_P THEN
      PA2:= 0;
      PA3:= 1;
      stable:= 0;
    END_IF;
    IF PA3 AND NOT PA4 AND TM_2_ta3.Q THEN
      PA3:= 0;
      PA4:= 1;
      stable:= 0;
    END_IF;

    (* Line B*)
    IF PB1 AND NOT PB2 AND TM_1_tb1.Q THEN
      PB1:= 0;
      PB2:= 1;
      stable:= 0;
    END_IF;
    IF PB2 AND NOT PB3 AND SB_P THEN
      PB2:= 0;
      PB3:= 1;
      stable:= 0;
    END_IF;
    IF PB3 AND NOT PB4 AND TM_2_tb3.Q THEN
      PB3:= 0;
      PB4:= 1;
      stable:= 0;
    END_IF;
    (* Line C *)
    IF PC1 AND NOT PC2 AND ST_Z THEN
      PC1:= 0;
      PC2:= 1;
      stable:= 0;
    END_IF;
    IF PC2 AND NOT PC3 AND NOT ST_Z THEN
      PC2:= 0;
      PC3:= 1;
      stable:= 0;
    END_IF;
    IF PC3 AND NOT PC4 AND TM_1_tc3.Q THEN
      PC3:= 0;
      PC4:= 1;
      stable:= 0;
    END_IF;
    IF PC4 AND NOT PC5 AND NOT SL_M THEN
      PC4:= 0;
      PC5:= 1;
      stable:= 0;
    END_IF;
    IF PC5 AND NOT PC6 AND ST_Z THEN
      PC5:= 0;
      PC6:= 1;
      stable:= 0;
    END_IF;
    (*HARD FIX *)
    IF TM_2_tc5.Q THEN
      PC5:= 0;
      PC7:= 1;
      stable:= 0;
    END_IF;
    IF PC6 AND NOT PC7 AND (NOT ST_Z OR TM_2_tc6.Q) THEN
      PC6:= 0;
      PC7:= 1;
      stable:= 0;
    END_IF;
    IF PC7 AND NOT PC8 AND ST_X THEN
      PC7:= 0;
      PC8:= 1;
      stable:= 0;
    END_IF;

    (* Line D *)
    IF PD1 AND NOT PD2 AND ST_Z THEN
      PD1:= 0;
      PD2:= 1;
      stable:= 0;
    END_IF;
    IF PD2 AND NOT PD3 AND NOT ST_Z THEN
      PD2:= 0;
      PD3:= 1;
      stable:= 0;
    END_IF;

    (* Line E *)
    IF PE1 AND NOT PE2 AND NOT SB_M THEN
      PE1:= 0;
      PE2:= 1;
      stable:= 0;
    END_IF;
    IF PE2 AND NOT PE3 AND NOT SBC THEN
      PE2:= 0;
      PE3:= 1;
      stable:= 0;
    END_IF;
    IF PE3 AND NOT PE4 AND SBC THEN
      PE3:= 0;
      PE4:= 1;
      stable:= 0;
    END_IF;
    IF PE4 AND NOT PE5 AND S_L THEN
      PE4:= 0;
      PE5:= 1;
      stable:= 0;
    END_IF;
    IF PE5 AND NOT PE6 AND NOT S_L THEN
      PE5:= 0;
      PE6:= 1;
      stable:= 0;
    END_IF;
    IF PE6 AND NOT PE7 AND NOT SBC THEN
      PE6:= 0;
      PE7:= 1;
      stable:= 0;
    END_IF;

    (* Line F *)
    IF PF1 AND NOT PF2 AND ST_Z THEN
      PF1:= 0;
      PF2:= 1;
      stable:= 0;
    END_IF;
    (*HARD FIX *)
    IF TM_2_tf1.Q THEN
      PF1:= 0;
      PF3:= 1;
      stable:= 0;
    END_IF;
    IF PF2 AND NOT PF3 AND (NOT ST_Z OR TM_2_tf2.Q) THEN
      PF2:= 0;
      PF3:= 1;
      stable:= 0;
    END_IF;
    IF PF3 AND NOT PF4 AND ST_X THEN
      PF3:= 0;
      PF4:= 1;
      stable:= 0;
    END_IF;
    IF PF4 AND NOT PF5 AND NOT ST_X THEN
      PF4:= 0;
      PF5:= 1;
      stable:= 0;
    END_IF;

    (* Across Lines *)
    IF PA4 AND PF5 AND NOT PC1 AND SL_M THEN
      PA4:= 0;
      PF5:= 0;
      PC1:= 1;
      stable:= 0;
    END_IF;
    IF PB4 AND PC8 AND NOT PD1 AND NOT ST_X AND SB_M THEN
      PB4:= 0;
      PC8:= 0;
      PD1:= 1;
      stable:= 0;
    END_IF;
    IF PD3 AND NOT PF1 AND NOT PE1 AND TM_1_td3.Q THEN
      PD3:= 0;
      PF1:= 1;
      PE1:= 1;
      stable:= 0;
    END_IF;
    IF PE7 AND NOT PA1 AND NOT PB1 AND SBC THEN
      PE7:= 0;
      PA1:= 1;
      PB1:= 1;
      stable:= 0;
    END_IF;

  (*============================================================*)
  (* OUTPUTS *)
  (*============================================================*)
  IF PA1 THEN
    AL_C:= 0;
  END_IF;
  IF PA2 OR PA3 THEN
    AL_C:= 1;
  END_IF;
  IF PA4 THEN
    AL_C:= 0;
    AL_M:= 1;
  END_IF;
  IF PB1 THEN
    AB_C:= 0;
  END_IF;
  IF PB2 OR PB3 THEN
    AB_C:= 1;
  END_IF;
  IF PB4 THEN
    AB_C:= 0;
    AB_M:= 1;
  END_IF;
  IF PC1 OR PC2 OR PD1 OR PD2 THEN
    AT_Z:= 1;
  END_IF;
  IF PC3 THEN
    AT_G:= 1;
  END_IF;
  IF PC4 THEN
    AL_M:= 0;
  END_IF;
  IF PC5 OR PC6 OR PF1 OR PF2 THEN
    AT_Z:= 0;
  END_IF;
  IF PC7 OR PC8 THEN
    AT_X:= 1;
  END_IF;
  IF PD3 THEN
    AT_G:= 0;
  END_IF;
  IF PE1 THEN
    AB_M:= 0;
  END_IF;
  IF PE2 OR PE3 THEN
    RB_M:= 1;
  END_IF;
  IF PE4 THEN
    AB_C:= 1;
  END_IF;
  IF PE5 THEN
    RB_M:= 1;
    AB_C:= 1;
  END_IF;
  IF PE6 OR PE7 THEN
    RB_M:= 0;
  END_IF;
  IF PF3 OR PF4 THEN
    AT_X:= 0;
  END_IF;
  IF PF5 THEN
    AT_X:= 0;
  END_IF;

END_PROGRAM

CONFIGURATION Config0

  RESOURCE Res0 ON PLC
    TASK task0(INTERVAL := T#20ms,PRIORITY := 0);
    PROGRAM instance0 WITH task0 : demo_factory;
  END_RESOURCE
END_CONFIGURATION

(* ---- production.st ---- *)
PROGRAM program0

(*=====================================================================*)
(*DECLARATION*)
(*=====================================================================*)

VAR

(*INPUTS*)
S_AL1_P_B1 AT %IX100.0 : BOOL;
S_AL1_P_B2 AT %IX100.1 : BOOL;
S_AL1_MCB AT %IX100.2 : BOOL;
MCB_BUSY AT %IX100.3 : BOOL;
S_AL1_MCBR AT %IX100.4 : BOOL;
MCBR_BUSY AT %IX100.5 : BOOL;
S_AL1_MCB2 AT %IX100.6 : BOOL;
S_AL1_MCBR2 AT %IX100.7 : BOOL;
E_AL1_B1 AT %QX100.0 : BOOL;
PUWS_AL1_B1_PLUS AT %QX100.1 : BOOL;
PUWS_AL1_B1_RIGHT AT %QX100.2 : BOOL;
PAS_AL1_PLUS AT %QX100.3 : BOOL;
PAS_AL1_TURN AT %QX100.4 : BOOL;

END_VAR

VAR

(*PLACES*)

PPAL1 : BOOL := 1;
PP0 : BOOL := 1;
PP1 : BOOL := 0;
PP2 : BOOL := 0;
PP3 : BOOL := 0;
PP4 : BOOL := 0;
MCB : BOOL := 1;
PP5 : BOOL := 0;
PP7 : BOOL := 0;
PPL3 : BOOL := 0;
PPL4 : BOOL := 0;
MCBR : BOOL := 1;
PPL5 : BOOL := 0;
PPL7 : BOOL := 0;
STABLE : BOOL := 0;

END_VAR

VAR

(*INTERNAL VARIABLES*)

MCB_CONTROL : BOOL;

END_VAR

(*=====================================================================*)
(*TRANSITIONS*)
(*=====================================================================*)

STABLE:=0;
WHILE STABLE=0 DO
   STABLE:=1;
   (*TP0*)
   IF (PP0) AND ( (NOT MCB_CONTROL) ) AND (NOT PP1) THEN
       PP0:=0;
       PP1:=1;
       STABLE:=0;
   END_IF;
   (*TP1*)
   IF (PP1) AND ( (S_AL1_P_B1) ) AND (NOT PP2) THEN
       PP1:=0;
       PP2:=1;
       STABLE:=0;
   END_IF;
   (*TP2*)
   IF (PP2) AND ( (S_AL1_P_B2 AND NOT MCB_CONTROL) ) AND (NOT PP3) THEN
       PP2:=0;
       PP3:=1;
       STABLE:=0;
   END_IF;
   (*TP3*)
   IF (PP3) AND ( (S_AL1_MCB) ) AND (NOT PP4 AND NOT PP1) THEN
       PP3:=0;
       PP4:=1;
       PP1:=1;
       STABLE:=0;
   END_IF;
   (*TP4*)
   IF (PP4 AND MCB) AND ( (MCB_BUSY) ) AND (NOT PP5) THEN
       PP4:=0;
       MCB:=0;
       PP5:=1;
       STABLE:=0;
   END_IF;
   (*TP6*)
   IF (PP5) AND ( (S_AL1_MCB2) ) AND (NOT PP7 AND NOT MCB) THEN
       PP5:=0;
       PP7:=1;
       MCB:=1;
       STABLE:=0;
   END_IF;
   (*TPL2*)
   IF (PP2) AND ( (S_AL1_P_B2 AND MCB_CONTROL) ) AND (NOT PPL3 AND NOT PP1) THEN
       PP2:=0;
       PPL3:=1;
       PP1:=1;
       STABLE:=0;
   END_IF;
   (*TPL3*)
   IF (PPL3) AND ( (S_AL1_MCBR) ) AND (NOT PPL4) THEN
       PPL3:=0;
       PPL4:=1;
       STABLE:=0;
   END_IF;
   (*TPL4*)
   IF (PPL4 AND MCBR) AND ( (MCBR_BUSY) ) AND (NOT PPL5) THEN
       PPL4:=0;
       MCBR:=0;
       PPL5:=1;
       STABLE:=0;
   END_IF;
   (*TPL6*)
   IF (PPL5) AND ( (S_AL1_MCBR2) ) AND (NOT PPL7 AND NOT MCBR) THEN
       PPL5:=0;
       PPL7:=1;
       MCBR:=1;
       STABLE:=0;
   END_IF;
END_WHILE;

(*=====================================================================*)
(*OUTPUTS*)
(*=====================================================================*)

(*E_AL1_B1*)
IF PP0 OR PP1 THEN
   E_AL1_B1:=1;
END_IF;
(*MCB_CONTROL*)
IF PP3 THEN
   MCB_CONTROL:=1;
END_IF;
(*PAS_AL1_PLUS*)
IF PPL3 OR PPL4 THEN
   PAS_AL1_PLUS:=1;
END_IF;
(*PAS_AL1_TURN*)
IF PPL3 OR PPL4 THEN
   PAS_AL1_TURN:=1;
END_IF;
(*PUWS_AL1_B1_PLUS*)
IF PPAL1 OR PP2 THEN
   PUWS_AL1_B1_PLUS:=1;
END_IF;
(*E_AL1_B1*)
IF PP2 OR PP3 OR PPL3 THEN
   E_AL1_B1:=0;
END_IF;
(*MCB_CONTROL*)
IF PP0 OR PPL3 THEN
   MCB_CONTROL:=0;
END_IF;
(*PAS_AL1_PLUS*)
IF PP0 OR PP3 OR PP4 THEN
   PAS_AL1_PLUS:=0;
END_IF;
(*PAS_AL1_TURN*)
IF PP0 OR PP3 OR PP4 THEN
   PAS_AL1_TURN:=0;
END_IF;
(*PUWS_AL1_B1_RIGHT*)
IF PPAL1 OR PP2 THEN
   PUWS_AL1_B1_RIGHT:=0;
END_IF;

END_PROGRAM

CONFIGURATION config0

    RESOURCE res0 ON PLC
        TASK task0(INTERVAL := T#20ms, PRIORITY := 0);
        PROGRAM instance0 WITH task0 : program0;
    END_RESOURCE

END_CONFIGURATION

(* ---- production_sorting_buffer_assembly.st ---- *)
PROGRAM program0

(*=====================================================================*)
(*DECLARATION*)
(*=====================================================================*)

VAR

(*INPUTS*)
S_AL1_P_B1 AT %IX102.5 : BOOL;
S_AL1_P_B2 AT %IX102.6 : BOOL;
S_AL1_MCB AT %IX102.7 : BOOL;
MCB_BUSY AT %IX103.0 : BOOL;
MCB_ERROR AT %IX103.1 : BOOL;
S_AL1_MCBR AT %IX103.2 : BOOL;
MCBR_BUSY AT %IX103.3 : BOOL;
MCBR_ERROR AT %IX103.4 : BOOL;
S_AL1_P_B3 AT %IX103.5 : BOOL;
S_AL1_MCB2 AT %IX103.6 : BOOL;
S_AL1_MCBR2 AT %IX103.7 : BOOL;
S_AL1_B AT %IX100.0 : BOOL;
P_AL1_B_FT AT %IX100.1 : BOOL;
P_AL1_B_BK AT %IX100.2 : BOOL;
S_AL1_B1 AT %IX100.3 : BOOL;
S_AL1_B2 AT %IX100.4 : BOOL;
S_AL1_B3 AT %IX100.5 : BOOL;
LP_AL1_CLAMPED AT %IX100.6 : BOOL;
S_AL1_LP AT %IX100.7 : BOOL;
S_AL1_L AT %IX101.0 : BOOL;
P_AL1_L_FT AT %IX101.1 : BOOL;
P_AL1_L_BK AT %IX101.2 : BOOL;
S_AL1_L1 AT %IX101.3 : BOOL;
S_AL1_L2 AT %IX101.4 : BOOL;
S_AL1_L3 AT %IX101.5 : BOOL;
RP_AL1_CLAMPED AT %IX101.6 : BOOL;
S_AL1_RP AT %IX101.7 : BOOL;
S_AL1 AT %IX102.0 : BOOL;
CS_AL1_W AT %IW100 : WORD;
S_BIN_1 AT %IX102.1 : BOOL;
S_AL1_BL AT %IX102.2 : BOOL;
AL1_DETECTED AT %IX102.3 : BOOL;
LP_AL1_LIMIT AT %IX102.4 : BOOL;
AL1_X_POS AT %IW101 : WORD;
AL1_Y_POS AT %IW102 : WORD;
AL1_Z_POS AT %IW103 : WORD;
S_AL1_ST1 AT %IX104.0 : BOOL;
S_AL1_ST2 AT %IX104.1 : BOOL;
S_AL1_ST3 AT %IX104.2 : BOOL;
RP_AL1_ST_CLAMPED AT %IX104.3 : BOOL;
AL1_ST_DETECTED AT %IX104.4 : BOOL;
AL1_ST_X_POS AT %IW104 : WORD;
AL1_ST_Y_POS AT %IW105 : WORD;
AL1_ST_Z_POS AT %IW106 : WORD;
E_AL1_B1 AT %QX102.0 : BOOL;
PUWS_AL1_B1_PLUS AT %QX102.1 : BOOL;
PUWS_AL1_B1_RIGHT AT %QX102.2 : BOOL;
PAS_AL1_PLUS AT %QX102.3 : BOOL;
PAS_AL1_TURN AT %QX102.4 : BOOL;
SB_AL1 AT %QX101.2 : BOOL;
PUWS_AL1_1_PLUS AT %QX101.3 : BOOL;
PUWS_AL1_1_RT AT %QX101.4 : BOOL;
CS_AL1_PLUS AT %QX101.5 : BOOL;
P_AL1_B AT %QX100.0 : BOOL;
SB_AL1_B1 AT %QX100.1 : BOOL;
SB_AL1_B2 AT %QX100.2 : BOOL;
SB_AL1_B3 AT %QX100.3 : BOOL;
LP_AL1_CLAMP AT %QX100.4 : BOOL;
P_AL1_L AT %QX100.5 : BOOL;
SB_AL1_L1 AT %QX100.6 : BOOL;
SB_AL1_L2 AT %QX100.7 : BOOL;
SB_AL1_L3 AT %QX101.0 : BOOL;
RP_AL1_CLAMP AT %QX101.1 : BOOL;
AL1_GRAB AT %QX101.6 : BOOL;
LP_AL1_RAISE AT %QX101.7 : BOOL;
AL1_X_SET AT %QW100 : WORD;
AL1_Y_SET AT %QW101 : WORD;
AL1_Z_SET AT %QW102 : WORD;
AL1_ST_X_SET AT %QW103 : WORD;
AL1_ST_Y_SET AT %QW104 : WORD;
AL1_ST_Z_SET AT %QW105 : WORD;
RP_AL1_ST_CLAMP AT %QX102.5 : BOOL;
AL1_ST_GRAB AT %QX102.6 : BOOL;
AL1_EMIT AT %QX102.7 : BOOL;
RC_AL1_ST AT %QX103.0 : BOOL;

END_VAR

VAR

(*PLACES*)

PPAL1 : BOOL := 1;
PP0 : BOOL := 1;
PP1 : BOOL := 0;
PP2 : BOOL := 0;
PP3 : BOOL := 0;
PP4 : BOOL := 0;
MCB : BOOL := 1;
PP5 : BOOL := 0;
PP7 : BOOL := 0;
PPL3 : BOOL := 0;
PPL4 : BOOL := 0;
MCBR : BOOL := 1;
PPL5 : BOOL := 0;
PPL7 : BOOL := 0;
P0 : BOOL := 1;
P1 : BOOL := 1;
P2 : BOOL := 0;
P3 : BOOL := 0;
P4 : BOOL := 0;
PB : BOOL := 0;
BIN1 : BOOL := 1;
BIN2 : BOOL := 0;
P5 : BOOL := 0;
P6 : BOOL := 0;
P_BASE : BOOL := 0;
PB1 : BOOL := 0;
PUSH_B : BOOL := 1;
PB2 : BOOL := 0;
PB23 : BOOL := 0;
PB3 : BOOL := 0;
PB4 : BOOL := 0;
PBF1 : BOOL := 1;
PB5 : BOOL := 0;
PBF2 : BOOL := 1;
PB6 : BOOL := 0;
PBF3 : BOOL := 1;
PB7 : BOOL := 0;
P_LID : BOOL := 0;
PL1 : BOOL := 0;
PUSH_L : BOOL := 1;
PL2 : BOOL := 0;
PL23 : BOOL := 0;
PL3 : BOOL := 0;
PL4 : BOOL := 0;
PLF1 : BOOL := 1;
PL5 : BOOL := 0;
PLF2 : BOOL := 1;
PL6 : BOOL := 0;
PLF3 : BOOL := 1;
PL7 : BOOL := 0;
PA0 : BOOL := 1;
PA1 : BOOL := 0;
PA2 : BOOL := 0;
PA3 : BOOL := 0;
PA4 : BOOL := 0;
PA5 : BOOL := 0;
PA6 : BOOL := 0;
PA7 : BOOL := 0;
PA8 : BOOL := 0;
PA9 : BOOL := 0;
PA10 : BOOL := 0;
PA11 : BOOL := 0;
PA12 : BOOL := 0;
PA13 : BOOL := 0;
PBF4 : BOOL := 1;
PB8 : BOOL := 0;
PB9 : BOOL := 0;
PLF4 : BOOL := 1;
PL8 : BOOL := 0;
PL9 : BOOL := 0;
PS0 : BOOL := 1;
PSC : BOOL := 1;
PS1 : BOOL := 0;
PS2 : BOOL := 0;
PS3 : BOOL := 0;
PS4 : BOOL := 0;
PS5 : BOOL := 0;
PS6 : BOOL := 0;
PS7 : BOOL := 0;
PS8 : BOOL := 0;
PS9 : BOOL := 0;
PS10 : BOOL := 0;
PS11 : BOOL := 0;
PS12 : BOOL := 0;
PSE1 : BOOL := 0;
PSE2 : BOOL := 0;
PSE0 : BOOL := 1;
STABLE : BOOL := 0;

END_VAR

VAR

(*INTERNAL VARIABLES*)

MCB_CONTROL : BOOL;
timer_1_TL1 : TON;
timer_1_TB1 : TON;
timer_1_P2 : TON;
timer_1_P3 : TON;
AL1_BASE : BOOL;
AL1_LID : BOOL;
timer_1_PL9 : TON;

END_VAR

timer_1_TL1(IN:= PL1, PT:= T#750ms);
timer_1_TB1(IN:= PB1, PT:= T#900ms);
timer_1_P2(IN:= P2, PT:= T#1000ms);
timer_1_P3(IN:= P3, PT:= T#1000ms);
timer_1_PL9(IN:= PL9, PT:= T#300ms);

(*=====================================================================*)
(*TRANSITIONS*)
(*=====================================================================*)

STABLE:=0;
WHILE STABLE=0 DO
   STABLE:=1;
   (*TP0*)
   IF (PP0) AND ( (NOT MCB_CONTROL) ) AND (NOT PP1) THEN
       PP0:=0;
       PP1:=1;
       STABLE:=0;
   END_IF;
   (*TP1*)
   IF (PP1) AND ( (S_AL1_P_B1) ) AND (NOT PP2) THEN
       PP1:=0;
       PP2:=1;
       STABLE:=0;
   END_IF;
   (*TP2*)
   IF (PP2) AND ( (S_AL1_P_B2 AND NOT MCB_CONTROL) ) AND (NOT PP3) THEN
       PP2:=0;
       PP3:=1;
       STABLE:=0;
   END_IF;
   (*TP3*)
   IF (PP3) AND ( (S_AL1_MCB) ) AND (NOT PP4 AND NOT PP1) THEN
       PP3:=0;
       PP4:=1;
       PP1:=1;
       STABLE:=0;
   END_IF;
   (*TP4*)
   IF (PP4 AND MCB) AND ( (MCB_BUSY) ) AND (NOT PP5) THEN
       PP4:=0;
       MCB:=0;
       PP5:=1;
       STABLE:=0;
   END_IF;
   (*TP6*)
   IF (PP5) AND ( (S_AL1_MCB2) ) AND (NOT PP7 AND NOT MCB) THEN
       PP5:=0;
       PP7:=1;
       MCB:=1;
       STABLE:=0;
   END_IF;
   (*TP7*)
   IF (PP7) AND ( (S_AL1_P_B3) ) AND (NOT P0) THEN
       PP7:=0;
       P0:=1;
       STABLE:=0;
   END_IF;
   (*TPL2*)
   IF (PP2) AND ( (S_AL1_P_B2 AND MCB_CONTROL) ) AND (NOT PPL3 AND NOT PP1) THEN
       PP2:=0;
       PPL3:=1;
       PP1:=1;
       STABLE:=0;
   END_IF;
   (*TPL3*)
   IF (PPL3) AND ( (S_AL1_MCBR) ) AND (NOT PPL4) THEN
       PPL3:=0;
       PPL4:=1;
       STABLE:=0;
   END_IF;
   (*TPL4*)
   IF (PPL4 AND MCBR) AND ( (MCBR_BUSY) ) AND (NOT PPL5) THEN
       PPL4:=0;
       MCBR:=0;
       PPL5:=1;
       STABLE:=0;
   END_IF;
   (*TPL6*)
   IF (PPL5) AND ( (S_AL1_MCBR2) ) AND (NOT PPL7 AND NOT MCBR) THEN
       PPL5:=0;
       PPL7:=1;
       MCBR:=1;
       STABLE:=0;
   END_IF;
   (*TPL7*)
   IF (PPL7) AND ( (S_AL1_P_B3) ) AND (NOT P0) THEN
       PPL7:=0;
       P0:=1;
       STABLE:=0;
   END_IF;
   (*T0212*)
   IF (P0 AND P1) AND ( (S_AL1) ) AND (NOT P2) THEN
       P0:=0;
       P1:=0;
       P2:=1;
       STABLE:=0;
   END_IF;
   (*T23*)
   IF (P2) AND ( (timer_1_P2.Q) ) AND (NOT P3) THEN
       P2:=0;
       P3:=1;
       STABLE:=0;
   END_IF;
   (*T34*)
   IF (P3) AND ( (timer_1_P3.Q) ) AND (NOT P4) THEN
       P3:=0;
       P4:=1;
       STABLE:=0;
   END_IF;
   (*T4B*)
   IF (P4) AND ( ((CS_AL1_W < 200) OR (CS_AL1_W > 400)) ) AND (NOT PB) THEN
       P4:=0;
       PB:=1;
       STABLE:=0;
   END_IF;
   (*T4B2*)
   IF (PB AND BIN1) AND ( (S_BIN_1) ) AND (NOT BIN2 AND NOT P1) THEN
       PB:=0;
       BIN1:=0;
       BIN2:=1;
       P1:=1;
       STABLE:=0;
   END_IF;
   (*TB21*)
   IF (BIN2) AND ( (NOT S_BIN_1) ) AND (NOT BIN1) THEN
       BIN2:=0;
       BIN1:=1;
       STABLE:=0;
   END_IF;
   (*T45*)
   IF (P4) AND ( ((CS_AL1_W > 200) AND (CS_AL1_W <= 300)) ) AND (NOT P5) THEN
       P4:=0;
       P5:=1;
       STABLE:=0;
   END_IF;
   (*T46*)
   IF (P4) AND ( ((CS_AL1_W > 300) AND (CS_AL1_W <= 400)) ) AND (NOT P6) THEN
       P4:=0;
       P6:=1;
       STABLE:=0;
   END_IF;
   (*T57*)
   IF (P5) AND ( (S_AL1_BL) ) AND (NOT P_LID AND NOT P1) THEN
       P5:=0;
       P_LID:=1;
       P1:=1;
       STABLE:=0;
   END_IF;
   (*T67*)
   IF (P6) AND ( (S_AL1_BL) ) AND (NOT P_BASE AND NOT P1) THEN
       P6:=0;
       P_BASE:=1;
       P1:=1;
       STABLE:=0;
   END_IF;
   (*TB0*)
   IF (P_BASE) AND ( (S_AL1_B) ) AND (NOT PB1) THEN
       P_BASE:=0;
       PB1:=1;
       STABLE:=0;
   END_IF;
   (*TB1*)
   IF (PB1 AND PUSH_B) AND ( (timer_1_TB1.Q) ) AND (NOT PB2) THEN
       PB1:=0;
       PUSH_B:=0;
       PB2:=1;
       STABLE:=0;
   END_IF;
   (*TB23*)
   IF (PB2) AND ( (P_AL1_B_FT) ) AND (NOT PB23) THEN
       PB2:=0;
       PB23:=1;
       STABLE:=0;
   END_IF;
   (*TB2*)
   IF (PB23) AND ( (P_AL1_B_FT) ) AND (NOT PB3) THEN
       PB23:=0;
       PB3:=1;
       STABLE:=0;
   END_IF;
   (*TB3*)
   IF (PB3) AND ( (P_AL1_B_BK) ) AND (NOT PB4 AND NOT PUSH_B) THEN
       PB3:=0;
       PB4:=1;
       PUSH_B:=1;
       STABLE:=0;
   END_IF;
   (*TB4*)
   IF (PB4 AND PBF1) AND ( (S_AL1_B1) ) AND (NOT PB5) THEN
       PB4:=0;
       PBF1:=0;
       PB5:=1;
       STABLE:=0;
   END_IF;
   (*TB5*)
   IF (PB5 AND PBF2) AND ( (S_AL1_B2) ) AND (NOT PB6 AND NOT PBF1) THEN
       PB5:=0;
       PBF2:=0;
       PB6:=1;
       PBF1:=1;
       STABLE:=0;
   END_IF;
   (*TB6*)
   IF (PB6 AND PBF3) AND ( (S_AL1_B3) ) AND (NOT PB7 AND NOT PBF2) THEN
       PB6:=0;
       PBF3:=0;
       PB7:=1;
       PBF2:=1;
       STABLE:=0;
   END_IF;
   (*TB7*)
   IF (PB7 AND PBF4) AND ( (S_AL1_LP) ) AND (NOT PB8) THEN
       PB7:=0;
       PBF4:=0;
       PB8:=1;
       STABLE:=0;
   END_IF;
   (*TL0*)
   IF (P_LID) AND ( (S_AL1_L) ) AND (NOT PL1) THEN
       P_LID:=0;
       PL1:=1;
       STABLE:=0;
   END_IF;
   (*TL1*)
   IF (PL1 AND PUSH_L) AND ( (timer_1_TL1.Q) ) AND (NOT PL2) THEN
       PL1:=0;
       PUSH_L:=0;
       PL2:=1;
       STABLE:=0;
   END_IF;
   (*TL23*)
   IF (PL2) AND ( (P_AL1_L_FT) ) AND (NOT PL23) THEN
       PL2:=0;
       PL23:=1;
       STABLE:=0;
   END_IF;
   (*TL2*)
   IF (PL23) AND ( (P_AL1_L_FT) ) AND (NOT PL3) THEN
       PL23:=0;
       PL3:=1;
       STABLE:=0;
   END_IF;
   (*TL3*)
   IF (PL3) AND ( (P_AL1_L_BK) ) AND (NOT PL4 AND NOT PUSH_L) THEN
       PL3:=0;
       PL4:=1;
       PUSH_L:=1;
       STABLE:=0;
   END_IF;
   (*TL4*)
   IF (PL4 AND PLF1) AND ( (S_AL1_L1) ) AND (NOT PL5) THEN
       PL4:=0;
       PLF1:=0;
       PL5:=1;
       STABLE:=0;
   END_IF;
   (*TL5*)
   IF (PL5 AND PLF2) AND ( (S_AL1_L2) ) AND (NOT PL6 AND NOT PLF1) THEN
       PL5:=0;
       PLF2:=0;
       PL6:=1;
       PLF1:=1;
       STABLE:=0;
   END_IF;
   (*TL6*)
   IF (PL6 AND PLF3) AND ( (S_AL1_L3) ) AND (NOT PL7 AND NOT PLF2) THEN
       PL6:=0;
       PLF3:=0;
       PL7:=1;
       PLF2:=1;
       STABLE:=0;
   END_IF;
   (*TL7*)
   IF (PL7 AND PLF4) AND ( (S_AL1_RP) ) AND (NOT PL8) THEN
       PL7:=0;
       PLF4:=0;
       PL8:=1;
       STABLE:=0;
   END_IF;
   (*TL8*)
   IF (PL8) AND ( (RP_AL1_CLAMPED) ) AND (NOT PL9) THEN
       PL8:=0;
       PL9:=1;
       STABLE:=0;
   END_IF;
   (*TB8*)
   IF (PB8) AND ( (LP_AL1_CLAMPED) ) AND (NOT PB9) THEN
       PB8:=0;
       PB9:=1;
       STABLE:=0;
   END_IF;
   (*TA0*)
   IF (PL9 AND PA0) AND ( (timer_1_PL9.Q AND RP_AL1_CLAMPED AND NOT AL1_DETECTED) ) AND (NOT PA1) THEN
       PL9:=0;
       PA0:=0;
       PA1:=1;
       STABLE:=0;
   END_IF;
   (*TA1*)
   IF (PA1) AND ( (AL1_X_POS>798 AND AL1_X_POS<802) ) AND (NOT PA2) THEN
       PA1:=0;
       PA2:=1;
       STABLE:=0;
   END_IF;
   (*TA2*)
   IF (PA2) AND ( (AL1_Z_POS>798 AND AL1_Z_POS<802) ) AND (NOT PA3) THEN
       PA2:=0;
       PA3:=1;
       STABLE:=0;
   END_IF;
   (*TA3*)
   IF (PA3) AND ( (NOT RP_AL1_CLAMPED) ) AND (NOT PA4) THEN
       PA3:=0;
       PA4:=1;
       STABLE:=0;
   END_IF;
   (*TA4*)
   IF (PA4) AND ( (AL1_Z_POS>398 AND AL1_Z_POS<402) ) AND (NOT PA5 AND NOT PLF3 AND NOT PLF4) THEN
       PA4:=0;
       PA5:=1;
       PLF3:=1;
       PLF4:=1;
       STABLE:=0;
   END_IF;
   (*TA5*)
   IF (PB9 AND PA5) AND ( (AL1_DETECTED AND LP_AL1_CLAMPED AND AL1_X_POS>208 AND AL1_X_POS<212) ) AND (NOT PA6) THEN
       PB9:=0;
       PA5:=0;
       PA6:=1;
       STABLE:=0;
   END_IF;
   (*TA6*)
   IF (PA6) AND ( (AL1_Z_POS>810 AND AL1_Z_POS<820) ) AND (NOT PA7) THEN
       PA6:=0;
       PA7:=1;
       STABLE:=0;
   END_IF;
   (*TA7*)
   IF (PA7) AND ( (AL1_Z_POS>398 AND AL1_Z_POS<402) ) AND (NOT PA8) THEN
       PA7:=0;
       PA8:=1;
       STABLE:=0;
   END_IF;
   (*TA8*)
   IF (PA8) AND ( (NOT LP_AL1_CLAMPED) ) AND (NOT PA9) THEN
       PA8:=0;
       PA9:=1;
       STABLE:=0;
   END_IF;
   (*TA9*)
   IF (PA9) AND ( (NOT LP_AL1_LIMIT) ) AND (NOT PA10) THEN
       PA9:=0;
       PA10:=1;
       STABLE:=0;
   END_IF;
   (*TA10*)
   IF (PA10) AND ( (LP_AL1_LIMIT) ) AND (NOT PA11) THEN
       PA10:=0;
       PA11:=1;
       STABLE:=0;
   END_IF;
   (*TA11*)
   IF (PA11) AND ( (NOT LP_AL1_LIMIT) ) AND (NOT PA12) THEN
       PA11:=0;
       PA12:=1;
       STABLE:=0;
   END_IF;
   (*TA12*)
   IF (PA12) AND ( (LP_AL1_LIMIT) ) AND (NOT PA13 AND NOT PA0 AND NOT PBF3 AND NOT PBF4) THEN
       PA12:=0;
       PA13:=1;
       PA0:=1;
       PBF3:=1;
       PBF4:=1;
       STABLE:=0;
   END_IF;
   (*TS1*)
   IF (PA13) AND ( (S_AL1_ST1) ) AND (NOT PS1) THEN
       PA13:=0;
       PS1:=1;
       STABLE:=0;
   END_IF;
   (*TS2*)
   IF (PS0 AND PSC AND PS1) AND ( (S_AL1_ST2) ) AND (NOT PS2) THEN
       PS0:=0;
       PSC:=0;
       PS1:=0;
       PS2:=1;
       STABLE:=0;
   END_IF;
   (*TS3*)
   IF (PS2) AND ( (RP_AL1_ST_CLAMPED) ) AND (NOT PS3) THEN
       PS2:=0;
       PS3:=1;
       STABLE:=0;
   END_IF;
   (*TS4*)
   IF (PS3) AND ( ((AL1_ST_Y_POS>540) AND (AL1_ST_Y_POS<580)) ) AND (NOT PS4) THEN
       PS3:=0;
       PS4:=1;
       STABLE:=0;
   END_IF;
   (*TS5*)
   IF (PS4) AND ( ((AL1_ST_Z_POS>730) AND (AL1_ST_Z_POS<770)) ) AND (NOT PSC AND NOT PS5) THEN
       PS4:=0;
       PSC:=1;
       PS5:=1;
       STABLE:=0;
   END_IF;
   (*TS6*)
   IF (PS5) AND ( (AL1_ST_DETECTED) ) AND (NOT PS6) THEN
       PS5:=0;
       PS6:=1;
       STABLE:=0;
   END_IF;
   (*TS7*)
   IF (PS6) AND ( ((AL1_ST_Z_POS>390) AND (AL1_ST_Z_POS<430)) ) AND (NOT PS7) THEN
       PS6:=0;
       PS7:=1;
       STABLE:=0;
   END_IF;
   (*TS8*)
   IF (PS7) AND ( ((AL1_ST_X_POS>840) AND (AL1_ST_X_POS<880)) ) AND (NOT PS8) THEN
       PS7:=0;
       PS8:=1;
       STABLE:=0;
   END_IF;
   (*TS9*)
   IF (PS8 AND PSE0) AND ( ((AL1_ST_Z_POS>580) AND (AL1_ST_Z_POS<620)) ) AND (NOT PS9) THEN
       PS8:=0;
       PSE0:=0;
       PS9:=1;
       STABLE:=0;
   END_IF;
   (*TS10*)
   IF (PS9) AND ( (NOT AL1_ST_DETECTED) ) AND (NOT PS0 AND NOT PS10 AND NOT PSE0) THEN
       PS9:=0;
       PS0:=1;
       PS10:=1;
       PSE0:=1;
       STABLE:=0;
   END_IF;
   (*TS11*)
   IF (PS9) AND ( (NOT AL1_ST_DETECTED) ) AND (NOT PS0 AND NOT PS11 AND NOT PSE0) THEN
       PS9:=0;
       PS0:=1;
       PS11:=1;
       PSE0:=1;
       STABLE:=0;
   END_IF;
   (*TS12*)
   IF (PS9) AND ( (NOT AL1_ST_DETECTED) ) AND (NOT PS0 AND NOT PS12 AND NOT PSE0) THEN
       PS9:=0;
       PS0:=1;
       PS12:=1;
       PSE0:=1;
       STABLE:=0;
   END_IF;
   (*TS13*)
   IF (PS10 AND PS11 AND PS12 AND PSE0) AND ( (TRUE) ) AND (NOT PSE1) THEN
       PS10:=0;
       PS11:=0;
       PS12:=0;
       PSE0:=0;
       PSE1:=1;
       STABLE:=0;
   END_IF;
   (*TSE1*)
   IF (PSE1) AND ( (NOT S_AL1_ST3) ) AND (NOT PSE2) THEN
       PSE1:=0;
       PSE2:=1;
       STABLE:=0;
   END_IF;
   (*TSE2*)
   IF (PSE2) AND ( (S_AL1_ST3) ) AND (NOT PSE0) THEN
       PSE2:=0;
       PSE0:=1;
       STABLE:=0;
   END_IF;
END_WHILE;

(*=====================================================================*)
(*OUTPUTS*)
(*=====================================================================*)

(*AL1_BASE*)
IF P6 THEN
   AL1_BASE:=1;
END_IF;
(*AL1_EMIT*)
IF PSE1 THEN
   AL1_EMIT:=1;
END_IF;
(*AL1_GRAB*)
IF PA3 OR PA4 OR PA5 OR PA6 THEN
   AL1_GRAB:=1;
END_IF;
(*AL1_LID*)
IF P5 THEN
   AL1_LID:=1;
END_IF;
(*AL1_ST_GRAB*)
IF PS5 OR PS6 OR PS7 OR PS8 THEN
   AL1_ST_GRAB:=1;
END_IF;
(*CS_AL1_PLUS*)
IF P1 OR P2 OR PB OR P5 OR P6 THEN
   CS_AL1_PLUS:=1;
END_IF;
(*E_AL1_B1*)
IF PP0 OR PP1 THEN
   E_AL1_B1:=1;
END_IF;
(*LP_AL1_CLAMP*)
IF PA6 OR PA7 OR PB8 OR PB9 THEN
   LP_AL1_CLAMP:=1;
END_IF;
(*LP_AL1_RAISE*)
IF PA9 OR PA10 THEN
   LP_AL1_RAISE:=1;
END_IF;
(*MCB_CONTROL*)
IF PP3 THEN
   MCB_CONTROL:=1;
END_IF;
(*PAS_AL1_PLUS*)
IF PPL3 OR PPL4 THEN
   PAS_AL1_PLUS:=1;
END_IF;
(*PAS_AL1_TURN*)
IF PPL3 OR PPL4 THEN
   PAS_AL1_TURN:=1;
END_IF;
(*PUWS_AL1_1_PLUS*)
IF PB OR P5 OR P6 THEN
   PUWS_AL1_1_PLUS:=1;
END_IF;
(*PUWS_AL1_1_RT*)
IF P5 OR P6 THEN
   PUWS_AL1_1_RT:=1;
END_IF;
(*PUWS_AL1_B1_PLUS*)
IF PPAL1 OR PP2 THEN
   PUWS_AL1_B1_PLUS:=1;
END_IF;
(*P_AL1_B*)
IF PB2 OR PB23 THEN
   P_AL1_B:=1;
END_IF;
(*P_AL1_L*)
IF PL2 OR PL23 THEN
   P_AL1_L:=1;
END_IF;
(*RC_AL1_ST*)
IF PSE1 OR PSE2 THEN
   RC_AL1_ST:=1;
END_IF;
(*RP_AL1_CLAMP*)
IF PL8 OR PL9 THEN
   RP_AL1_CLAMP:=1;
END_IF;
(*RP_AL1_ST_CLAMP*)
IF PS2 OR PS3 OR PS4 THEN
   RP_AL1_ST_CLAMP:=1;
END_IF;
(*SB_AL1*)
IF P3 OR P4 OR PB OR P5 OR P6 THEN
   SB_AL1:=1;
END_IF;
(*SB_AL1_B1*)
IF PB5 THEN
   SB_AL1_B1:=1;
END_IF;
(*SB_AL1_B2*)
IF PB6 THEN
   SB_AL1_B2:=1;
END_IF;
(*SB_AL1_B3*)
IF PB7 THEN
   SB_AL1_B3:=1;
END_IF;
(*SB_AL1_L1*)
IF PL5 THEN
   SB_AL1_L1:=1;
END_IF;
(*SB_AL1_L2*)
IF PL6 THEN
   SB_AL1_L2:=1;
END_IF;
(*SB_AL1_L3*)
IF PL7 THEN
   SB_AL1_L3:=1;
END_IF;
(*AL1_BASE*)
IF P1 OR P5 THEN
   AL1_BASE:=0;
END_IF;
(*AL1_EMIT*)
IF PSE2 OR PSE0 THEN
   AL1_EMIT:=0;
END_IF;
(*AL1_GRAB*)
IF PA0 OR PA1 OR PA2 OR PA7 OR PA8 THEN
   AL1_GRAB:=0;
END_IF;
(*AL1_LID*)
IF P1 OR P6 THEN
   AL1_LID:=0;
END_IF;
(*AL1_ST_GRAB*)
IF PS2 OR PS3 OR PS4 OR PS9 THEN
   AL1_ST_GRAB:=0;
END_IF;
(*CS_AL1_PLUS*)
IF P3 OR P4 THEN
   CS_AL1_PLUS:=0;
END_IF;
(*E_AL1_B1*)
IF PP2 OR PP3 OR PPL3 THEN
   E_AL1_B1:=0;
END_IF;
(*LP_AL1_CLAMP*)
IF PA8 OR PA9 OR PA10 OR PA11 OR PA12 OR PBF4 THEN
   LP_AL1_CLAMP:=0;
END_IF;
(*LP_AL1_RAISE*)
IF PA0 OR PA1 OR PA2 OR PA3 OR PA4 OR PA5 OR PA6 OR PA7 OR PA8 OR PA11 OR PA12 THEN
   LP_AL1_RAISE:=0;
END_IF;
(*MCB_CONTROL*)
IF PP0 OR PPL3 THEN
   MCB_CONTROL:=0;
END_IF;
(*PAS_AL1_PLUS*)
IF PP0 OR PP3 OR PP4 THEN
   PAS_AL1_PLUS:=0;
END_IF;
(*PAS_AL1_TURN*)
IF PP0 OR PP3 OR PP4 THEN
   PAS_AL1_TURN:=0;
END_IF;
(*PUWS_AL1_1_PLUS*)
IF P1 OR P2 OR P3 OR P4 THEN
   PUWS_AL1_1_PLUS:=0;
END_IF;
(*PUWS_AL1_1_RT*)
IF P1 OR P2 OR P3 OR P4 OR PB THEN
   PUWS_AL1_1_RT:=0;
END_IF;
(*PUWS_AL1_B1_RIGHT*)
IF PPAL1 OR PP2 THEN
   PUWS_AL1_B1_RIGHT:=0;
END_IF;
(*P_AL1_B*)
IF P_BASE OR PB1 OR PB3 THEN
   P_AL1_B:=0;
END_IF;
(*P_AL1_L*)
IF P_LID OR PL1 OR PL3 THEN
   P_AL1_L:=0;
END_IF;
(*RC_AL1_ST*)
IF PSE0 THEN
   RC_AL1_ST:=0;
END_IF;
(*RP_AL1_CLAMP*)
IF PA3 OR PA4 OR PLF4 THEN
   RP_AL1_CLAMP:=0;
END_IF;
(*RP_AL1_ST_CLAMP*)
IF PSC THEN
   RP_AL1_ST_CLAMP:=0;
END_IF;
(*SB_AL1*)
IF P1 OR P2 THEN
   SB_AL1:=0;
END_IF;
(*SB_AL1_B1*)
IF PBF1 THEN
   SB_AL1_B1:=0;
END_IF;
(*SB_AL1_B2*)
IF PBF2 THEN
   SB_AL1_B2:=0;
END_IF;
(*SB_AL1_B3*)
IF PBF3 THEN
   SB_AL1_B3:=0;
END_IF;
(*SB_AL1_L1*)
IF PLF1 THEN
   SB_AL1_L1:=0;
END_IF;
(*SB_AL1_L2*)
IF PLF2 THEN
   SB_AL1_L2:=0;
END_IF;
(*SB_AL1_L3*)
IF PLF3 THEN
   SB_AL1_L3:=0;
END_IF;
(*AL1_X_SET*)
IF PA0 THEN
   AL1_X_SET:=210;
END_IF;
(*AL1_X_SET*)
IF PA1 THEN
   AL1_X_SET:=800;
END_IF;
(*AL1_Z_SET*)
IF PA2 THEN
   AL1_Z_SET:=800;
END_IF;
(*AL1_Z_SET*)
IF PA4 THEN
   AL1_Z_SET:=400;
END_IF;
(*AL1_X_SET*)
IF PA5 THEN
   AL1_X_SET:=210;
END_IF;
(*AL1_Z_SET*)
IF PA6 THEN
   AL1_Z_SET:=818;
END_IF;
(*AL1_Z_SET*)
IF PA7 THEN
   AL1_Z_SET:=400;
END_IF;
(*AL1_ST_X_SET*)
IF PS0 THEN
   AL1_ST_X_SET:=0;
END_IF;
(*AL1_ST_Y_SET*)
IF PS3 THEN
   AL1_ST_Y_SET:=560;
END_IF;
(*AL1_ST_Z_SET*)
IF PS4 THEN
   AL1_ST_Z_SET:=750;
END_IF;
(*AL1_ST_Z_SET*)
IF PS6 THEN
   AL1_ST_Z_SET:=410;
END_IF;
(*AL1_ST_X_SET*)
IF PS7 THEN
   AL1_ST_X_SET:=860;
END_IF;
(*AL1_ST_Z_SET*)
IF PS8 THEN
   AL1_ST_Z_SET:=600;
END_IF;

END_PROGRAM

CONFIGURATION config0

    RESOURCE res0 ON PLC
        TASK task0(INTERVAL := T#20ms, PRIORITY := 0);
        PROGRAM instance0 WITH task0 : program0;
    END_RESOURCE

END_CONFIGURATION

(* ---- stacking.st ---- *)
PROGRAM program0

(*=====================================================================*)
(*DECLARATION*)
(*=====================================================================*)

VAR

(*INPUTS*)
S_AL1_ST1 AT %IX100.0 : BOOL;
S_AL1_ST2 AT %IX100.1 : BOOL;
S_AL1_ST3 AT %IX100.2 : BOOL;
RP_AL1_ST_CLAMPED AT %IX100.3 : BOOL;
AL1_ST_DETECTED AT %IX100.4 : BOOL;
RESET AT %IX100.5 : BOOL;
AL1_ST_X_POS AT %IW100 : WORD;
AL1_ST_Y_POS AT %IW101 : WORD;
AL1_ST_Z_POS AT %IW102 : WORD;
RUNNING AT %IX100.7 : BOOL;
AL1_ST_X_SET AT %QW100 : WORD;
AL1_ST_Y_SET AT %QW101 : WORD;
AL1_ST_Z_SET AT %QW102 : WORD;
RP_AL1_ST_CLAMP AT %QX100.0 : BOOL;
AL1_ST_GRAB AT %QX100.1 : BOOL;
AL1_EMIT AT %QX100.2 : BOOL;
RC_AL1_ST AT %QX100.3 : BOOL;

END_VAR

VAR

(*PLACES*)

PA13 : BOOL := 1;
PS0 : BOOL := 1;
PSC : BOOL := 1;
PS1 : BOOL := 0;
PS2 : BOOL := 0;
PS3 : BOOL := 0;
PS4 : BOOL := 0;
PS5 : BOOL := 0;
PS6 : BOOL := 0;
PS7 : BOOL := 0;
PS8 : BOOL := 0;
PS9 : BOOL := 0;
PS10 : BOOL := 0;
PS11 : BOOL := 0;
PS12 : BOOL := 0;
PSE1 : BOOL := 0;
PSE2 : BOOL := 0;
PSE0 : BOOL := 1;
STABLE : BOOL := 0;

END_VAR

(*=====================================================================*)
(*TRANSITIONS*)
(*=====================================================================*)

STABLE:=0;
WHILE STABLE=0 DO
   STABLE:=1;
   (*TS1*)
   IF (PA13) AND ( (S_AL1_ST1) ) AND (NOT PS1) THEN
       PA13:=0;
       PS1:=1;
       STABLE:=0;
   END_IF;
   (*TS2*)
   IF (PS0 AND PSC AND PS1) AND ( (S_AL1_ST2) ) AND (NOT PS2) THEN
       PS0:=0;
       PSC:=0;
       PS1:=0;
       PS2:=1;
       STABLE:=0;
   END_IF;
   (*TS3*)
   IF (PS2) AND ( (RP_AL1_ST_CLAMPED) ) AND (NOT PS3) THEN
       PS2:=0;
       PS3:=1;
       STABLE:=0;
   END_IF;
   (*TS4*)
   IF (PS3) AND ( ((AL1_ST_Y_POS>540) AND (AL1_ST_Y_POS<580)) ) AND (NOT PS4) THEN
       PS3:=0;
       PS4:=1;
       STABLE:=0;
   END_IF;
   (*TS5*)
   IF (PS4) AND ( ((AL1_ST_Z_POS>730) AND (AL1_ST_Z_POS<770)) ) AND (NOT PSC AND NOT PS5) THEN
       PS4:=0;
       PSC:=1;
       PS5:=1;
       STABLE:=0;
   END_IF;
   (*TS6*)
   IF (PS5) AND ( (AL1_ST_DETECTED) ) AND (NOT PS6) THEN
       PS5:=0;
       PS6:=1;
       STABLE:=0;
   END_IF;
   (*TS7*)
   IF (PS6) AND ( ((AL1_ST_Z_POS>390) AND (AL1_ST_Z_POS<430)) ) AND (NOT PS7) THEN
       PS6:=0;
       PS7:=1;
       STABLE:=0;
   END_IF;
   (*TS8*)
   IF (PS7) AND ( ((AL1_ST_X_POS>840) AND (AL1_ST_X_POS<880)) ) AND (NOT PS8) THEN
       PS7:=0;
       PS8:=1;
       STABLE:=0;
   END_IF;
   (*TS9*)
   IF (PS8 AND PSE0) AND ( ((AL1_ST_Z_POS>580) AND (AL1_ST_Z_POS<620)) ) AND (NOT PS9) THEN
       PS8:=0;
       PSE0:=0;
       PS9:=1;
       STABLE:=0;
   END_IF;
   (*TS10*)
   IF (PS9) AND ( (NOT AL1_ST_DETECTED) ) AND (NOT PS0 AND NOT PS10 AND NOT PSE0 AND NOT PA13) THEN
       PS9:=0;
       PS0:=1;
       PS10:=1;
       PSE0:=1;
       PA13:=1;
       STABLE:=0;
   END_IF;
   (*TS11*)
   IF (PS9) AND ( (NOT AL1_ST_DETECTED) ) AND (NOT PS0 AND NOT PS11 AND NOT PSE0 AND NOT PA13) THEN
       PS9:=0;
       PS0:=1;
       PS11:=1;
       PSE0:=1;
       PA13:=1;
       STABLE:=0;
   END_IF;
   (*TS12*)
   IF (PS9) AND ( (NOT AL1_ST_DETECTED) ) AND (NOT PS0 AND NOT PS12 AND NOT PSE0 AND NOT PA13) THEN
       PS9:=0;
       PS0:=1;
       PS12:=1;
       PSE0:=1;
       PA13:=1;
       STABLE:=0;
   END_IF;
   (*TS13*)
   IF (PS10 AND PS11 AND PS12 AND PSE0) AND ( (TRUE) ) AND (NOT PSE1) THEN
       PS10:=0;
       PS11:=0;
       PS12:=0;
       PSE0:=0;
       PSE1:=1;
       STABLE:=0;
   END_IF;
   (*TSE1*)
   IF (PSE1) AND ( (NOT S_AL1_ST3) ) AND (NOT PSE2) THEN
       PSE1:=0;
       PSE2:=1;
       STABLE:=0;
   END_IF;
   (*TSE2*)
   IF (PSE2) AND ( (S_AL1_ST3) ) AND (NOT PSE0) THEN
       PSE2:=0;
       PSE0:=1;
       STABLE:=0;
   END_IF;
END_WHILE;

(*=====================================================================*)
(*OUTPUTS*)
(*=====================================================================*)

(*AL1_EMIT*)
IF PSE1 THEN
   AL1_EMIT:=1;
END_IF;
(*AL1_ST_GRAB*)
IF PS5 OR PS6 OR PS7 OR PS8 THEN
   AL1_ST_GRAB:=1;
END_IF;
(*RC_AL1_ST*)
IF PSE1 OR PSE2 THEN
   RC_AL1_ST:=1;
END_IF;
(*RP_AL1_ST_CLAMP*)
IF PS2 OR PS3 OR PS4 THEN
   RP_AL1_ST_CLAMP:=1;
END_IF;
(*AL1_EMIT*)
IF PSE2 OR PSE0 THEN
   AL1_EMIT:=0;
END_IF;
(*AL1_ST_GRAB*)
IF PS2 OR PS3 OR PS4 OR PS9 THEN
   AL1_ST_GRAB:=0;
END_IF;
(*RC_AL1_ST*)
IF PSE0 THEN
   RC_AL1_ST:=0;
END_IF;
(*RP_AL1_ST_CLAMP*)
IF PSC THEN
   RP_AL1_ST_CLAMP:=0;
END_IF;
(*AL1_ST_X_SET*)
IF PS0 THEN
   AL1_ST_X_SET:=0;
END_IF;
(*AL1_ST_Y_SET*)
IF PS3 THEN
   AL1_ST_Y_SET:=560;
END_IF;
(*AL1_ST_Z_SET*)
IF PS4 THEN
   AL1_ST_Z_SET:=750;
END_IF;
(*AL1_ST_Z_SET*)
IF PS6 THEN
   AL1_ST_Z_SET:=410;
END_IF;
(*AL1_ST_X_SET*)
IF PS7 THEN
   AL1_ST_X_SET:=860;
END_IF;
(*AL1_ST_Z_SET*)
IF PS8 THEN
   AL1_ST_Z_SET:=600;
END_IF;

END_PROGRAM

CONFIGURATION config0

    RESOURCE res0 ON PLC
        TASK task0(INTERVAL := T#20ms, PRIORITY := 0);
        PROGRAM instance0 WITH task0 : program0;
    END_RESOURCE

END_CONFIGURATION

(* ---- storage_model.st ---- *)
PROGRAM program0

(*=====================================================================*)
(*DECLARATION*)
(*=====================================================================*)

VAR

(*INPUTS*)
AL1_G_S1 AT %IX100.0 : BOOL;
AL1_G_SC_LL AT %IX100.1 : BOOL;
AL1_G_SC_MZ AT %IX100.2 : BOOL;
AL1_G_ML AT %IX100.3 : BOOL;
AL1_G_SC_MX AT %IX100.4 : BOOL;
AL1_G_SC_RL AT %IX100.5 : BOOL;
RC_AL1_G7 AT %QX100.0 : BOOL;
AL1_G_SC_LT AT %QX100.1 : BOOL;
AL1_G_SC_LIFT AT %QX100.2 : BOOL;
AL1_G_SC_RT AT %QX100.3 : BOOL;
AL1_G_SC_TG AT %QW100 : INT;

END_VAR

VAR

(*PLACES*)

PG : BOOL := 1;
PG1 : BOOL := 0;
PG2 : BOOL := 0;
PG3 : BOOL := 0;
PG4 : BOOL := 0;
PG5 : BOOL := 0;
PG6 : BOOL := 0;
PG7 : BOOL := 0;
PG8 : BOOL := 0;
PG9 : BOOL := 0;
PG10 : BOOL := 0;
PG11 : BOOL := 0;
PG12 : BOOL := 0;
PG13 : BOOL := 0;
PG14 : BOOL := 0;
PG15 : BOOL := 0;
PG16 : BOOL := 0;
PG17 : BOOL := 0;
PG18 : BOOL := 0;
PG19 : BOOL := 0;
PG20 : BOOL := 0;
PG21 : BOOL := 0;
PG22 : BOOL := 0;
PG23 : BOOL := 0;
PG24 : BOOL := 0;
PG25 : BOOL := 0;
PG26 : BOOL := 0;
STABLE : BOOL := 0;

END_VAR

VAR

(*INTERNAL VARIABLES*)

TG_POS : INT;

END_VAR

TG_POS:=10;

(*=====================================================================*)
(*TRANSITIONS*)
(*=====================================================================*)

STABLE:=0;
WHILE STABLE=0 DO
   STABLE:=1;
   (*TG1*)
   IF (PG) AND ( (NOT AL1_G_S1) ) AND (NOT PG1) THEN
       PG:=0;
       PG1:=1;
       STABLE:=0;
   END_IF;
   (*TG2*)
   IF (PG1) AND ( (AL1_G_SC_LL) ) AND (NOT PG2) THEN
       PG1:=0;
       PG2:=1;
       STABLE:=0;
   END_IF;
   (*TG3*)
   IF (PG2) AND ( (AL1_G_SC_MZ) ) AND (NOT PG3) THEN
       PG2:=0;
       PG3:=1;
       STABLE:=0;
   END_IF;
   (*TG4*)
   IF (PG3) AND ( (NOT AL1_G_SC_MZ) ) AND (NOT PG4) THEN
       PG3:=0;
       PG4:=1;
       STABLE:=0;
   END_IF;
   (*TG5*)
   IF (PG4) AND ( (AL1_G_ML) ) AND (NOT PG5) THEN
       PG4:=0;
       PG5:=1;
       STABLE:=0;
   END_IF;
   (*TG6*)
   IF (PG5) AND ( (AL1_G_SC_MZ) ) AND (NOT PG6) THEN
       PG5:=0;
       PG6:=1;
       STABLE:=0;
   END_IF;
   (*TG7*)
   IF (PG6) AND ( (NOT AL1_G_SC_MZ) ) AND (NOT PG7) THEN
       PG6:=0;
       PG7:=1;
       STABLE:=0;
   END_IF;
   (*TG8*)
   IF (PG7) AND ( (TRUE) ) AND (NOT PG8 AND NOT PG11) THEN
       PG7:=0;
       PG8:=1;
       PG11:=1;
       STABLE:=0;
   END_IF;
   (*TG9*)
   IF (PG8) AND ( (AL1_G_SC_MX) ) AND (NOT PG9) THEN
       PG8:=0;
       PG9:=1;
       STABLE:=0;
   END_IF;
   (*TG10*)
   IF (PG9) AND ( (NOT AL1_G_SC_MX) ) AND (NOT PG10) THEN
       PG9:=0;
       PG10:=1;
       STABLE:=0;
   END_IF;
   (*TG12*)
   IF (PG11) AND ( (AL1_G_SC_MZ) ) AND (NOT PG12) THEN
       PG11:=0;
       PG12:=1;
       STABLE:=0;
   END_IF;
   (*TG13*)
   IF (PG12) AND ( (NOT AL1_G_SC_MZ) ) AND (NOT PG13) THEN
       PG12:=0;
       PG13:=1;
       STABLE:=0;
   END_IF;
   (*TG14*)
   IF (PG10 AND PG13) AND ( (TRUE) ) AND (NOT PG14) THEN
       PG10:=0;
       PG13:=0;
       PG14:=1;
       STABLE:=0;
   END_IF;
   (*TG15*)
   IF (PG14) AND ( (AL1_G_SC_MZ) ) AND (NOT PG15) THEN
       PG14:=0;
       PG15:=1;
       STABLE:=0;
   END_IF;
   (*TG16*)
   IF (PG15) AND ( (NOT AL1_G_SC_MZ) ) AND (NOT PG16) THEN
       PG15:=0;
       PG16:=1;
       STABLE:=0;
   END_IF;
   (*TG17*)
   IF (PG16) AND ( (AL1_G_SC_RL) ) AND (NOT PG17) THEN
       PG16:=0;
       PG17:=1;
       STABLE:=0;
   END_IF;
   (*TG18*)
   IF (PG17) AND ( (AL1_G_SC_MZ) ) AND (NOT PG18) THEN
       PG17:=0;
       PG18:=1;
       STABLE:=0;
   END_IF;
   (*TG19*)
   IF (PG18) AND ( (NOT AL1_G_SC_MZ) ) AND (NOT PG19) THEN
       PG18:=0;
       PG19:=1;
       STABLE:=0;
   END_IF;
   (*TG20*)
   IF (PG19) AND ( (AL1_G_ML) ) AND (NOT PG20) THEN
       PG19:=0;
       PG20:=1;
       STABLE:=0;
   END_IF;
   (*TG21*)
   IF (PG20) AND ( (TRUE) ) AND (NOT PG21 AND NOT PG24) THEN
       PG20:=0;
       PG21:=1;
       PG24:=1;
       STABLE:=0;
   END_IF;
   (*TG22*)
   IF (PG21) AND ( (AL1_G_SC_MX) ) AND (NOT PG22) THEN
       PG21:=0;
       PG22:=1;
       STABLE:=0;
   END_IF;
   (*TG23*)
   IF (PG22) AND ( (NOT AL1_G_SC_MX) ) AND (NOT PG23) THEN
       PG22:=0;
       PG23:=1;
       STABLE:=0;
   END_IF;
   (*TG25*)
   IF (PG24) AND ( (AL1_G_SC_MZ) ) AND (NOT PG25) THEN
       PG24:=0;
       PG25:=1;
       STABLE:=0;
   END_IF;
   (*TG26*)
   IF (PG25) AND ( (NOT AL1_G_SC_MZ) ) AND (NOT PG26) THEN
       PG25:=0;
       PG26:=1;
       STABLE:=0;
   END_IF;
   (*TG27*)
   IF (PG23 AND PG26) AND ( (TRUE) ) AND (NOT PG) THEN
       PG23:=0;
       PG26:=0;
       PG:=1;
       STABLE:=0;
   END_IF;
END_WHILE;

(*=====================================================================*)
(*OUTPUTS*)
(*=====================================================================*)

(*AL1_G_SC_LIFT*)
IF PG2 OR PG3 OR PG4 OR PG14 OR PG15 OR PG16 THEN
   AL1_G_SC_LIFT:=1;
END_IF;
(*AL1_G_SC_LT*)
IF PG1 OR PG2 OR PG3 THEN
   AL1_G_SC_LT:=1;
END_IF;
(*AL1_G_SC_RT*)
IF PG16 OR PG17 OR PG18 THEN
   AL1_G_SC_RT:=1;
END_IF;
(*RC_AL1_G7*)
IF PG THEN
   RC_AL1_G7:=1;
END_IF;
(*AL1_G_SC_LIFT*)
IF PG OR PG1 OR PG5 OR PG6 OR PG7 OR PG8 OR PG9 OR PG10 OR PG11 OR PG12 OR PG13 OR PG17 OR PG18 OR PG19 OR PG20 OR PG21 OR PG22 OR PG23 OR PG24 OR PG25 OR PG26 THEN
   AL1_G_SC_LIFT:=0;
END_IF;
(*AL1_G_SC_LT*)
IF PG OR PG4 OR PG5 OR PG6 OR PG7 OR PG8 OR PG9 OR PG10 OR PG11 OR PG12 OR PG13 OR PG14 OR PG15 OR PG16 OR PG17 OR PG18 OR PG19 OR PG20 OR PG21 OR PG22 OR PG23 OR PG24 OR PG25 OR PG26 THEN
   AL1_G_SC_LT:=0;
END_IF;
(*AL1_G_SC_RT*)
IF PG OR PG1 OR PG2 OR PG3 OR PG4 OR PG5 OR PG6 OR PG7 OR PG8 OR PG9 OR PG10 OR PG11 OR PG12 OR PG13 OR PG14 OR PG15 OR PG19 OR PG20 OR PG21 OR PG22 OR PG23 OR PG24 OR PG25 OR PG26 THEN
   AL1_G_SC_RT:=0;
END_IF;
(*RC_AL1_G7*)
IF PG1 OR PG2 OR PG3 OR PG4 OR PG5 OR PG6 OR PG7 OR PG8 OR PG9 OR PG10 OR PG11 OR PG12 OR PG13 OR PG14 OR PG15 OR PG16 OR PG17 OR PG18 OR PG19 OR PG20 OR PG21 OR PG22 OR PG23 OR PG24 OR PG25 OR PG26 THEN
   RC_AL1_G7:=0;
END_IF;
(*AL1_G_SC_TG*)
IF PG THEN
   AL1_G_SC_TG:=55;
END_IF;
(*AL1_G_SC_TG*)
IF PG1 THEN
   AL1_G_SC_TG:=55;
END_IF;
(*AL1_G_SC_TG*)
IF PG2 THEN
   AL1_G_SC_TG:=55;
END_IF;
(*AL1_G_SC_TG*)
IF PG3 THEN
   AL1_G_SC_TG:=55;
END_IF;
(*AL1_G_SC_TG*)
IF PG4 THEN
   AL1_G_SC_TG:=55;
END_IF;
(*AL1_G_SC_TG*)
IF PG5 THEN
   AL1_G_SC_TG:=55;
END_IF;
(*AL1_G_SC_TG*)
IF PG6 THEN
   AL1_G_SC_TG:=55;
END_IF;
(*AL1_G_SC_TG*)
IF PG7 THEN
   AL1_G_SC_TG:=TG_POS;
END_IF;
(*AL1_G_SC_TG*)
IF PG8 THEN
   AL1_G_SC_TG:=TG_POS;
END_IF;
(*AL1_G_SC_TG*)
IF PG9 THEN
   AL1_G_SC_TG:=TG_POS;
END_IF;
(*AL1_G_SC_TG*)
IF PG10 THEN
   AL1_G_SC_TG:=TG_POS;
END_IF;
(*AL1_G_SC_TG*)
IF PG11 THEN
   AL1_G_SC_TG:=TG_POS;
END_IF;
(*AL1_G_SC_TG*)
IF PG12 THEN
   AL1_G_SC_TG:=TG_POS;
END_IF;
(*AL1_G_SC_TG*)
IF PG13 THEN
   AL1_G_SC_TG:=TG_POS;
END_IF;
(*AL1_G_SC_TG*)
IF PG14 THEN
   AL1_G_SC_TG:=TG_POS;
END_IF;
(*AL1_G_SC_TG*)
IF PG15 THEN
   AL1_G_SC_TG:=TG_POS;
END_IF;
(*AL1_G_SC_TG*)
IF PG16 THEN
   AL1_G_SC_TG:=TG_POS;
END_IF;
(*AL1_G_SC_TG*)
IF PG17 THEN
   AL1_G_SC_TG:=TG_POS;
END_IF;
(*AL1_G_SC_TG*)
IF PG18 THEN
   AL1_G_SC_TG:=TG_POS;
END_IF;
(*AL1_G_SC_TG*)
IF PG19 THEN
   AL1_G_SC_TG:=TG_POS;
END_IF;
(*AL1_G_SC_TG*)
IF PG20 THEN
   AL1_G_SC_TG:=55;
END_IF;
(*AL1_G_SC_TG*)
IF PG21 THEN
   AL1_G_SC_TG:=55;
END_IF;
(*AL1_G_SC_TG*)
IF PG22 THEN
   AL1_G_SC_TG:=55;
END_IF;
(*AL1_G_SC_TG*)
IF PG23 THEN
   AL1_G_SC_TG:=55;
END_IF;
(*AL1_G_SC_TG*)
IF PG24 THEN
   AL1_G_SC_TG:=55;
END_IF;
(*AL1_G_SC_TG*)
IF PG25 THEN
   AL1_G_SC_TG:=55;
END_IF;
(*AL1_G_SC_TG*)
IF PG26 THEN
   AL1_G_SC_TG:=55;
END_IF;

END_PROGRAM

CONFIGURATION config0

    RESOURCE res0 ON PLC
        TASK task0(INTERVAL := T#20ms, PRIORITY := 0);
        PROGRAM instance0 WITH task0 : program0;
    END_RESOURCE

END_CONFIGURATION
